C01805=1100.666,-5.311,447.503,176.248,14.221,151.801
C01806=1100.661,-5.561,447.516,176.246,14.220,151.802
C01807=1100.655,-5.810,447.530,176.244,14.220,151.802
C01808=1100.649,-6.060,447.543,176.242,14.219,151.803
C01809=1100.643,-6.309,447.557,176.240,14.219,151.803
C01810=1100.637,-6.559,447.571,176.238,14.218,151.803
C01811=1100.631,-6.808,447.584,176.236,14.218,151.804
C01812=1100.626,-7.058,447.597,176.234,14.218,151.804
C01813=1100.620,-7.307,447.610,176.232,14.217,151.804
C01814=1100.614,-7.557,447.624,176.230,14.216,151.805
C01815=1100.608,-7.806,447.637,176.228,14.216,151.805
C01816=1100.602,-8.055,447.651,176.225,14.215,151.805
C01817=1100.597,-8.306,447.664,176.223,14.214,151.806
C01818=1100.590,-8.555,447.677,176.221,14.214,151.806
C01819=1100.585,-8.804,447.691,176.219,14.213,151.807
C01820=1100.578,-9.054,447.705,176.217,14.213,151.807
C01821=1100.573,-9.305,447.718,176.215,14.212,151.807
C01822=1100.567,-9.554,447.731,176.213,14.211,151.808
C01823=1100.561,-9.804,447.745,176.210,14.211,151.808
C01824=1100.555,-10.053,447.758,176.208,14.211,151.808
C01825=1100.550,-10.303,447.771,176.206,14.210,151.809
C01826=1100.544,-10.552,447.785,176.204,14.210,151.809
C01827=1100.537,-10.801,447.798,176.202,14.209,151.809
C01828=1100.532,-11.052,447.811,176.200,14.209,151.810
C01829=1100.526,-11.301,447.824,176.198,14.208,151.810
C01830=1100.521,-11.551,447.838,176.195,14.207,151.810
C01831=1100.515,-11.800,447.851,176.193,14.206,151.811
C01832=1100.509,-12.050,447.864,176.191,14.206,151.811
C01833=1100.503,-12.299,447.878,176.189,14.205,151.811
C01834=1100.498,-12.548,447.890,176.187,14.205,151.812
C01835=1100.492,-12.798,447.904,176.185,14.204,151.812
C01836=1100.486,-13.047,447.917,176.183,14.204,151.813
C01837=1100.480,-13.297,447.930,176.181,14.203,151.813
C01838=1100.475,-13.547,447.944,176.179,14.203,151.813
C01839=1100.468,-13.796,447.957,176.177,14.202,151.813
C01840=1100.463,-14.046,447.970,176.175,14.201,151.814
C01841=1100.457,-14.295,447.983,176.173,14.201,151.814
C01842=1100.451,-14.545,447.996,176.171,14.200,151.815
C01843=1100.446,-14.795,448.010,176.169,14.200,151.815
C01844=1100.440,-15.045,448.022,176.167,14.199,151.815
C01845=1100.434,-15.294,448.035,176.165,14.198,151.816
C01846=1100.428,-15.544,448.049,176.163,14.198,151.816
C01847=1100.422,-15.794,448.062,176.160,14.197,151.816
C01848=1100.416,-16.061,448.076,176.158,14.196,151.817
C01849=1100.409,-16.328,448.090,176.156,14.196,151.817
C01850=1100.403,-16.596,448.104,176.154,14.195,151.817
C01851=1100.397,-16.863,448.118,176.152,14.195,151.818
C01852=1100.391,-17.113,448.131,176.150,14.194,151.818
C01853=1100.385,-17.362,448.144,176.148,14.194,151.818
C01854=1100.379,-17.612,448.157,176.145,14.194,151.819
C01855=1100.373,-17.861,448.170,176.144,14.193,151.819
C01856=1100.367,-18.111,448.183,176.141,14.193,151.820
C01857=1100.362,-18.360,448.196,176.140,14.192,151.820
C01858=1100.356,-18.610,448.209,176.137,14.191,151.820
C01859=1100.350,-18.859,448.222,176.135,14.190,151.821
C01860=1100.344,-19.109,448.235,176.133,14.190,151.821
C01861=1100.338,-19.358,448.248,176.131,14.189,151.821
C01862=1100.333,-19.609,448.261,176.128,14.189,151.822
C01863=1100.327,-19.858,448.274,176.127,14.188,151.822
C01864=1100.321,-20.108,448.287,176.125,14.187,151.822
C01865=1100.315,-20.358,448.299,176.123,14.187,151.823
C01866=1100.309,-20.607,448.313,176.121,14.186,151.823
C01867=1100.303,-20.857,448.325,176.118,14.186,151.823
C01868=1100.298,-21.106,448.339,176.117,14.185,151.824
C01869=1100.292,-21.356,448.351,176.114,14.185,151.824
C01870=1100.286,-21.606,448.364,176.113,14.184,151.824
C01871=1100.280,-21.855,448.377,176.110,14.184,151.825
C01872=1100.274,-22.105,448.390,176.108,14.183,151.825
C01873=1100.268,-22.354,448.403,176.106,14.183,151.825
C01874=1100.262,-22.604,448.416,176.104,14.182,151.826
C01875=1100.257,-22.853,448.428,176.102,14.181,151.826
C01876=1100.251,-23.103,448.442,176.100,14.181,151.826
C01877=1100.245,-23.352,448.454,176.098,14.180,151.827
C01878=1100.239,-23.602,448.467,176.096,14.180,151.827
C01879=1100.233,-23.852,448.480,176.094,14.179,151.827
C01880=1100.227,-24.101,448.492,176.092,14.178,151.828
C01881=1100.221,-24.351,448.505,176.090,14.178,151.828
C01882=1100.215,-24.600,448.518,176.088,14.177,151.828
C01883=1100.210,-24.850,448.531,176.086,14.177,151.829
C01884=1100.204,-25.100,448.544,176.084,14.176,151.829
C01885=1100.198,-25.350,448.556,176.082,14.176,151.829
C01886=1100.192,-25.599,448.569,176.080,14.175,151.830
C01887=1100.187,-25.848,448.582,176.078,14.174,151.830
C01888=1100.181,-26.098,448.594,176.076,14.174,151.830
C01889=1100.175,-26.348,448.607,176.074,14.173,151.831
C01890=1100.169,-26.597,448.620,176.072,14.173,151.831
C01891=1100.163,-26.847,448.633,176.070,14.172,151.831
C01892=1100.158,-27.096,448.645,176.068,14.172,151.832
C01893=1100.152,-27.346,448.657,176.066,14.171,151.832
C01894=1100.146,-27.596,448.671,176.064,14.170,151.832
C01895=1100.140,-27.845,448.683,176.062,14.170,151.833
C01896=1100.134,-28.095,448.696,176.060,14.169,151.833
C01897=1100.128,-28.345,448.708,176.058,14.169,151.833
C01898=1100.123,-28.594,448.720,176.056,14.168,151.834
C01899=1100.116,-28.844,448.734,176.054,14.168,151.834
C01900=1100.110,-29.094,448.746,176.052,14.167,151.834
C01901=1100.105,-29.343,448.759,176.050,14.166,151.835
C01902=1100.099,-29.593,448.771,176.048,14.166,151.835
C01903=1100.093,-29.842,448.784,176.046,14.165,151.835
C01904=1100.087,-30.092,448.796,176.044,14.165,151.836
C01905=1100.080,-30.341,448.809,176.042,14.164,151.836
C01906=1100.075,-30.591,448.821,176.040,14.164,151.836
C01907=1100.069,-30.841,448.834,176.038,14.163,151.837
C01908=1100.063,-31.090,448.846,176.036,14.162,151.837
C01909=1100.057,-31.340,448.859,176.034,14.162,151.837
C01910=1100.052,-31.590,448.871,176.032,14.161,151.838
C01911=1100.046,-31.840,448.884,176.030,14.161,151.838
C01912=1100.039,-32.106,448.896,176.028,14.160,151.838
C01913=1100.033,-32.372,448.911,176.026,14.160,151.839
C01914=1100.026,-32.639,448.924,176.024,14.159,151.839
C01915=1100.021,-32.906,448.937,176.022,14.158,151.839
C01916=1100.015,-33.156,448.950,176.020,14.158,151.840
C01917=1100.008,-33.405,448.962,176.018,14.157,151.840
C01918=1100.003,-33.654,448.974,176.016,14.157,151.840
C01919=1099.997,-33.904,448.986,176.014,14.156,151.841
C01920=1099.991,-34.154,448.999,176.012,14.156,151.841
C01921=1099.985,-34.404,449.011,176.010,14.155,151.841
C01922=1099.980,-34.653,449.024,176.008,14.154,151.842
C01923=1099.973,-34.903,449.036,176.006,14.154,151.842
C01924=1099.967,-35.153,449.048,176.004,14.153,151.842
C01925=1099.962,-35.402,449.060,176.002,14.153,151.843
C01926=1099.956,-35.652,449.073,176.000,14.152,151.843
C01927=1099.950,-35.902,449.085,175.998,14.152,151.843
C01928=1099.944,-36.152,449.098,175.996,14.151,151.844
C01929=1099.938,-36.400,449.110,175.994,14.151,151.844
C01930=1099.932,-36.650,449.122,175.993,14.150,151.844
C01931=1099.927,-36.900,449.135,175.991,14.150,151.844
C01932=1099.921,-37.149,449.147,175.989,14.149,151.845
C01933=1099.915,-37.399,449.159,175.987,14.148,151.845
C01934=1099.909,-37.649,449.172,175.985,14.148,151.845
C01935=1099.903,-37.898,449.184,175.983,14.147,151.846
C01936=1099.897,-38.148,449.196,175.981,14.147,151.846
C01937=1099.892,-38.398,449.209,175.978,14.146,151.847
C01938=1099.887,-38.648,449.220,175.977,14.146,151.847
C01939=1099.880,-38.897,449.232,175.975,14.145,151.847
C01940=1099.874,-39.147,449.245,175.973,14.144,151.848
C01941=1099.869,-39.396,449.257,175.971,14.144,151.848
C01942=1099.862,-39.646,449.269,175.969,14.143,151.848
C01943=1099.856,-39.896,449.281,175.967,14.143,151.848
C01944=1099.851,-40.145,449.294,175.965,14.142,151.849
C01945=1099.844,-40.394,449.306,175.963,14.142,151.849
C01946=1099.838,-40.644,449.318,175.961,14.141,151.849
C01947=1099.833,-40.894,449.330,175.959,14.141,151.850
C01948=1099.827,-41.144,449.342,175.957,14.140,151.850
C01949=1099.821,-41.394,449.354,175.956,14.140,151.850
C01950=1099.815,-41.643,449.366,175.953,14.139,151.851
C01951=1099.809,-41.892,449.378,175.951,14.139,151.851
C01952=1099.803,-42.142,449.391,175.950,14.138,151.851
C01953=1099.797,-42.392,449.402,175.947,14.137,151.852
C01954=1099.791,-42.642,449.414,175.945,14.137,151.852
C01955=1099.785,-42.891,449.427,175.943,14.136,151.852
C01956=1099.779,-43.140,449.438,175.941,14.136,151.853
C01957=1099.773,-43.390,449.451,175.940,14.135,151.853
C01958=1099.768,-43.641,449.463,175.938,14.135,151.853
C01959=1099.762,-43.890,449.474,175.936,14.134,151.854
C01960=1099.756,-44.139,449.487,175.934,14.134,151.854
C01961=1099.750,-44.388,449.498,175.932,14.133,151.854
C01962=1099.744,-44.639,449.510,175.930,14.133,151.855
C01963=1099.738,-44.889,449.523,175.928,14.132,151.855
C01964=1099.732,-45.138,449.534,175.926,14.131,151.855
C01965=1099.726,-45.387,449.547,175.924,14.131,151.856
C01966=1099.720,-45.638,449.558,175.922,14.130,151.856
C01967=1099.715,-45.887,449.570,175.920,14.130,151.856
C01968=1099.708,-46.136,449.582,175.919,14.130,151.856
C01969=1099.703,-46.386,449.594,175.917,14.129,151.857
C01970=1099.697,-46.636,449.606,175.915,14.128,151.857
C01971=1099.691,-46.885,449.618,175.913,14.128,151.858
C01972=1099.685,-47.135,449.630,175.911,14.127,151.858
C01973=1099.679,-47.385,449.642,175.909,14.127,151.858
C01974=1099.673,-47.634,449.654,175.907,14.126,151.859
C01975=1099.667,-47.884,449.665,175.905,14.126,151.859
C01976=1099.661,-48.151,449.678,175.903,14.125,151.859
C01977=1099.655,-48.419,449.691,175.901,14.124,151.859
C01978=1099.649,-48.685,449.704,175.899,14.124,151.860
C01979=1099.643,-48.952,449.716,175.897,14.123,151.860
C01980=1099.637,-49.202,449.728,175.895,14.123,151.860
C01981=1099.630,-49.451,449.740,175.893,14.122,151.861
C01982=1099.625,-49.701,449.752,175.892,14.122,151.861
C01983=1099.618,-49.951,449.764,175.890,14.121,151.861
C01984=1099.613,-50.200,449.775,175.888,14.121,151.862
C01985=1099.607,-50.450,449.787,175.886,14.120,151.862
C01986=1099.601,-50.699,449.799,175.884,14.120,151.862
C01987=1099.595,-50.949,449.811,175.882,14.119,151.863
C01988=1099.589,-51.198,449.822,175.880,14.119,151.863
C01989=1099.583,-51.449,449.834,175.878,14.118,151.863
C01990=1099.577,-51.698,449.846,175.877,14.118,151.864
C01991=1099.571,-51.948,449.857,175.875,14.117,151.864
C01992=1099.565,-52.198,449.870,175.873,14.117,151.864
C01993=1099.559,-52.447,449.881,175.871,14.116,151.865
C01994=1099.553,-52.697,449.892,175.868,14.116,151.865
C01995=1099.546,-52.946,449.904,175.867,14.115,151.865
C01996=1099.541,-53.196,449.916,175.865,14.114,151.866
C01997=1099.534,-53.446,449.928,175.863,14.115,151.866
C01998=1099.529,-53.695,449.939,175.861,14.114,151.866
C01999=1099.523,-53.945,449.951,175.859,14.114,151.867
C02000=1099.517,-54.195,449.962,175.857,14.113,151.867
C02001=1099.510,-54.444,449.974,175.855,14.112,151.867
C02002=1099.505,-54.694,449.985,175.853,14.112,151.868
C02003=1099.499,-54.944,449.997,175.851,14.111,151.868
C02004=1099.492,-55.194,450.009,175.850,14.111,151.868
C02005=1099.486,-55.443,450.020,175.848,14.111,151.869
C02006=1099.481,-55.693,450.032,175.846,14.110,151.869
C02007=1099.475,-55.942,450.044,175.844,14.110,151.869
C02008=1099.468,-56.192,450.055,175.842,14.109,151.870
C02009=1099.462,-56.441,450.067,175.840,14.109,151.870
C02010=1099.457,-56.692,450.078,175.839,14.108,151.870
C02011=1099.451,-56.941,450.089,175.837,14.108,151.870
C02012=1099.444,-57.191,450.101,175.835,14.107,151.871
C02013=1099.439,-57.440,450.112,175.833,14.107,151.871
C02014=1099.433,-57.690,450.125,175.831,14.106,151.872
C02015=1099.427,-57.939,450.136,175.829,14.106,151.872
C02016=1099.421,-58.190,450.147,175.828,14.105,151.872
C02017=1099.415,-58.438,450.158,175.825,14.105,151.872
C02018=1099.408,-58.689,450.170,175.824,14.104,151.873
C02019=1099.403,-58.938,450.182,175.821,14.104,151.873
C02020=1099.397,-59.188,450.193,175.820,14.103,151.873
C02021=1099.391,-59.438,450.204,175.818,14.103,151.874
C02022=1099.384,-59.687,450.216,175.816,14.103,151.874
C02023=1099.379,-59.937,450.227,175.814,14.102,151.874
C02024=1099.373,-60.187,450.239,175.812,14.102,151.875
C02025=1099.367,-60.436,450.250,175.810,14.101,151.875
C02026=1099.361,-60.685,450.261,175.808,14.100,151.875
C02027=1099.355,-60.936,450.272,175.807,14.101,151.876
C02028=1099.349,-61.185,450.284,175.805,14.100,151.876
C02029=1099.343,-61.435,450.296,175.803,14.099,151.876
C02030=1099.337,-61.685,450.307,175.801,14.099,151.877
C02031=1099.331,-61.934,450.319,175.799,14.098,151.877
C02032=1099.325,-62.184,450.329,175.798,14.098,151.877
C02033=1099.319,-62.434,450.341,175.796,14.098,151.878
C02034=1099.314,-62.684,450.352,175.794,14.097,151.878
C02035=1099.308,-62.932,450.364,175.792,14.097,151.878
C02036=1099.301,-63.183,450.375,175.790,14.096,151.879
C02037=1099.296,-63.432,450.386,175.788,14.095,151.879
C02038=1099.289,-63.682,450.397,175.787,14.095,151.879
C02039=1099.283,-63.931,450.409,175.785,14.095,151.879
C02040=1099.278,-64.200,450.421,175.783,14.094,151.880
C02041=1099.271,-64.468,450.433,175.781,14.094,151.880
C02042=1099.264,-64.736,450.446,175.778,14.093,151.881
C02043=1099.258,-65.005,450.457,175.777,14.093,151.881
C02044=1099.252,-65.254,450.468,175.775,14.092,151.881
C02045=1099.246,-65.504,450.479,175.773,14.092,151.882
C02046=1099.240,-65.754,450.490,175.771,14.091,151.882
C02047=1099.235,-66.003,450.502,175.769,14.091,151.882
C02048=1099.228,-66.253,450.514,175.767,14.090,151.883
C02049=1099.223,-66.503,450.525,175.765,14.090,151.883
C02050=1099.217,-66.752,450.535,175.764,14.090,151.883
C02051=1099.210,-67.002,450.547,175.762,14.089,151.883
C02052=1099.205,-67.252,450.558,175.760,14.088,151.884
C02053=1099.198,-67.501,450.570,175.758,14.088,151.884
C02054=1099.192,-67.751,450.580,175.757,14.088,151.884
C02055=1099.187,-68.000,450.591,175.755,14.088,151.885
C02056=1099.181,-68.251,450.603,175.753,14.087,151.885
C02057=1099.175,-68.500,450.614,175.751,14.086,151.885
C02058=1099.170,-68.750,450.625,175.749,14.086,151.886
C02059=1099.163,-69.000,450.636,175.748,14.086,151.886
C02060=1099.157,-69.250,450.647,175.746,14.085,151.886
C02061=1099.152,-69.499,450.658,175.744,14.085,151.887
C02062=1099.145,-69.749,450.670,175.742,14.084,151.887
C02063=1099.139,-69.998,450.681,175.741,14.084,151.887
C02064=1099.134,-70.248,450.692,175.738,14.083,151.888
C02065=1099.128,-70.497,450.702,175.737,14.083,151.888
C02066=1099.121,-70.747,450.714,175.734,14.082,151.888
C02067=1099.116,-70.997,450.725,175.733,14.082,151.889
C02068=1099.110,-71.246,450.735,175.731,14.081,151.889
C02069=1099.104,-71.496,450.747,175.729,14.081,151.889
C02070=1099.098,-71.746,450.758,175.727,14.080,151.889
C02071=1099.093,-71.996,450.769,175.725,14.080,151.890
C02072=1099.087,-72.245,450.780,175.724,14.080,151.890
C02073=1099.081,-72.495,450.791,175.722,14.079,151.890
C02074=1099.075,-72.745,450.802,175.720,14.078,151.891
C02075=1099.069,-72.994,450.813,175.718,14.078,151.891
C02076=1099.063,-73.245,450.824,175.717,14.078,151.891
C02077=1099.057,-73.494,450.835,175.715,14.077,151.892
C02078=1099.052,-73.744,450.846,175.713,14.077,151.892
C02079=1099.046,-73.993,450.857,175.711,14.076,151.892
C02080=1099.039,-74.243,450.868,175.710,14.077,151.893
C02081=1099.034,-74.493,450.879,175.708,14.076,151.893
C02082=1099.028,-74.742,450.890,175.706,14.075,151.893
C02083=1099.022,-74.991,450.900,175.704,14.075,151.894
C02084=1099.015,-75.242,450.911,175.703,14.075,151.894
C02085=1099.009,-75.491,450.922,175.700,14.074,151.894
C02086=1099.004,-75.741,450.933,175.698,14.074,151.895
C02087=1098.997,-75.991,450.944,175.697,14.074,151.895
C02088=1098.992,-76.240,450.955,175.695,14.073,151.895
C02089=1098.986,-76.490,450.966,175.693,14.072,151.896
C02090=1098.979,-76.740,450.977,175.691,14.072,151.896
C02091=1098.973,-76.990,450.987,175.690,14.072,151.896
C02092=1098.968,-77.239,450.998,175.688,14.072,151.897
C02093=1098.962,-77.489,451.009,175.686,14.071,151.897
C02094=1098.956,-77.739,451.020,175.685,14.071,151.897
C02095=1098.950,-77.988,451.031,175.683,14.071,151.898
C02096=1098.943,-78.238,451.041,175.681,14.070,151.898
C02097=1098.938,-78.487,451.052,175.678,14.070,151.898
C02098=1098.931,-78.737,451.063,175.677,14.069,151.898
C02099=1098.926,-78.987,451.074,175.675,14.069,151.899
C02100=1098.920,-79.237,451.084,175.673,14.068,151.899
C02101=1098.914,-79.486,451.095,175.672,14.068,151.899
C02102=1098.907,-79.736,451.106,175.670,14.068,151.900
C02103=1098.902,-79.986,451.117,175.668,14.067,151.900
C02104=1098.895,-80.256,451.129,175.666,14.067,151.901
C02105=1098.889,-80.527,451.140,175.664,14.066,151.901
C02106=1098.882,-80.797,451.151,175.663,14.066,151.901
C02107=1098.875,-81.068,451.163,175.660,14.066,151.902
C02108=1098.870,-81.318,451.174,175.658,14.065,151.902
C02109=1098.863,-81.567,451.184,175.656,14.065,151.902
C02110=1098.857,-81.817,451.195,175.655,14.065,151.903
C02111=1098.851,-82.066,451.206,175.653,14.065,151.903
C02112=1098.845,-82.316,451.216,175.651,14.064,151.903
C02113=1098.839,-82.566,451.227,175.650,14.064,151.904
C02114=1098.832,-82.816,451.237,175.648,14.064,151.904
C02115=1098.826,-83.065,451.248,175.646,14.063,151.904
C02116=1098.821,-83.315,451.258,175.644,14.063,151.905
C02117=1098.814,-83.564,451.269,175.643,14.062,151.905
C02118=1098.808,-83.815,451.280,175.640,14.062,151.905
C02119=1098.802,-84.064,451.291,175.639,14.062,151.906
C02120=1098.796,-84.314,451.300,175.637,14.062,151.906
C02121=1098.790,-84.563,451.311,175.635,14.061,151.906
C02122=1098.784,-84.814,451.322,175.634,14.061,151.907
C02123=1098.778,-85.063,451.333,175.632,14.061,151.907
C02124=1098.772,-85.313,451.343,175.630,14.060,151.907
C02125=1098.766,-85.562,451.353,175.629,14.060,151.908
C02126=1098.760,-85.811,451.364,175.626,14.060,151.908
C02127=1098.754,-86.062,451.375,175.625,14.059,151.908
C02128=1098.748,-86.311,451.385,175.623,14.059,151.909
C02129=1098.742,-86.561,451.396,175.621,14.059,151.909
C02130=1098.735,-86.810,451.406,175.619,14.058,151.909
C02131=1098.730,-87.060,451.416,175.618,14.058,151.910
C02132=1098.724,-87.310,451.427,175.616,14.058,151.910
C02133=1098.717,-87.560,451.438,175.614,14.057,151.910
C02134=1098.712,-87.810,451.448,175.612,14.058,151.911
C02135=1098.705,-88.059,451.458,175.610,14.057,151.911
C02136=1098.699,-88.308,451.469,175.608,14.057,151.911
C02137=1098.693,-88.559,451.480,175.607,14.056,151.912
C02138=1098.687,-88.808,451.490,175.605,14.056,151.912
C02139=1098.681,-89.058,451.500,175.603,14.055,151.912
C02140=1098.675,-89.308,451.510,175.602,14.056,151.913
C02141=1098.669,-89.557,451.521,175.600,14.055,151.913
C02142=1098.663,-89.807,451.531,175.598,14.055,151.913
C02143=1098.657,-90.056,451.542,175.596,14.055,151.914
C02144=1098.651,-90.307,451.552,175.594,14.054,151.914
C02145=1098.645,-90.556,451.562,175.593,14.054,151.914
C02146=1098.639,-90.806,451.573,175.591,14.054,151.915
C02147=1098.633,-91.056,451.583,175.589,14.053,151.915
C02148=1098.627,-91.305,451.594,175.588,14.053,151.915
C02149=1098.621,-91.555,451.603,175.586,14.053,151.916
C02150=1098.615,-91.804,451.614,175.584,14.052,151.916
C02151=1098.608,-92.055,451.624,175.582,14.052,151.916
C02152=1098.603,-92.304,451.635,175.580,14.052,151.917
C02153=1098.596,-92.554,451.645,175.578,14.051,151.917
C02154=1098.591,-92.804,451.655,175.577,14.052,151.917
C02155=1098.584,-93.053,451.666,175.575,14.051,151.918
C02156=1098.579,-93.303,451.676,175.574,14.051,151.918
C02157=1098.573,-93.553,451.687,175.572,14.050,151.918
C02158=1098.567,-93.802,451.696,175.570,14.050,151.919
C02159=1098.561,-94.052,451.707,175.568,14.050,151.919
C02160=1098.554,-94.302,451.717,175.566,14.050,151.919
C02161=1098.549,-94.552,451.728,175.564,14.049,151.920
C02162=1098.543,-94.802,451.738,175.563,14.049,151.920
C02163=1098.537,-95.051,451.748,175.561,14.049,151.920
C02164=1098.531,-95.301,451.758,175.560,14.049,151.921
C02165=1098.525,-95.550,451.769,175.558,14.048,151.921
C02166=1098.519,-95.800,451.778,175.555,14.048,151.921
C02167=1098.513,-96.050,451.789,175.554,14.048,151.922
C02168=1098.506,-96.323,451.799,175.552,14.048,151.922
C02169=1098.500,-96.595,451.811,175.550,14.047,151.922
C02170=1098.493,-96.868,451.822,175.549,14.047,151.923
C02171=1098.486,-97.141,451.833,175.547,14.047,151.923
C02172=1098.481,-97.391,451.844,175.545,14.046,151.923
C02173=1098.474,-97.640,451.854,175.543,14.046,151.924
C02174=1098.469,-97.890,451.864,175.541,14.046,151.924
C02175=1098.463,-98.140,451.874,175.539,14.045,151.925
C02176=1098.456,-98.389,451.884,175.538,14.045,151.925
C02177=1098.451,-98.640,451.894,175.536,14.045,151.925
C02178=1098.444,-98.889,451.904,175.535,14.045,151.926
C02179=1098.438,-99.138,451.914,175.533,14.045,151.926
C02180=1098.433,-99.389,451.924,175.530,14.044,151.926
C02181=1098.426,-99.638,451.934,175.529,14.044,151.927
C02182=1098.420,-99.888,451.944,175.527,14.044,151.927
C02183=1098.413,-100.137,451.955,175.526,14.044,151.927
C02184=1098.408,-100.388,451.965,175.524,14.044,151.928
C02185=1098.401,-100.637,451.974,175.522,14.044,151.928
C02186=1098.395,-100.887,451.985,175.520,14.043,151.928
C02187=1098.389,-101.137,451.995,175.518,14.043,151.929
C02188=1098.383,-101.386,452.004,175.517,14.043,151.929
C02189=1098.377,-101.636,452.015,175.515,14.042,151.929
C02190=1098.371,-101.886,452.025,175.514,14.043,151.930
C02191=1098.365,-102.136,452.034,175.512,14.042,151.930
C02192=1098.359,-102.385,452.045,175.510,14.042,151.931
C02193=1098.353,-102.634,452.054,175.508,14.042,151.931
C02194=1098.347,-102.885,452.064,175.506,14.041,151.931
C02195=1098.341,-103.134,452.075,175.505,14.041,151.931
C02196=1098.334,-103.384,452.084,175.503,14.041,151.932
C02197=1098.329,-103.634,452.094,175.501,14.041,151.932
C02198=1098.323,-103.883,452.104,175.499,14.041,151.933
C02199=1098.316,-104.133,452.114,175.498,14.041,151.933
C02200=1098.310,-104.382,452.124,175.496,14.040,151.933
C02201=1098.305,-104.633,452.134,175.495,14.041,151.934
C02202=1098.298,-104.882,452.144,175.493,14.040,151.934
C02203=1098.292,-105.132,452.154,175.491,14.040,151.934
C02204=1098.286,-105.381,452.163,175.489,14.040,151.935
C02205=1098.280,-105.631,452.173,175.487,14.039,151.935
C02206=1098.274,-105.881,452.184,175.486,14.039,151.935
C02207=1098.268,-106.130,452.193,175.484,14.039,151.936
C02208=1098.262,-106.380,452.203,175.483,14.039,151.936
C02209=1098.256,-106.630,452.212,175.480,14.039,151.936
C02210=1098.250,-106.880,452.223,175.479,14.039,151.937
C02211=1098.244,-107.129,452.233,175.477,14.038,151.937
C02212=1098.237,-107.379,452.242,175.476,14.039,151.938
C02213=1098.231,-107.629,452.252,175.474,14.038,151.938
C02214=1098.225,-107.879,452.262,175.472,14.038,151.938
C02215=1098.219,-108.129,452.271,175.470,14.038,151.939
C02216=1098.213,-108.378,452.282,175.468,14.037,151.939
C02217=1098.207,-108.628,452.292,175.467,14.038,151.939
C02218=1098.201,-108.878,452.301,175.465,14.037,151.940
C02219=1098.195,-109.127,452.311,175.463,14.037,151.940
C02220=1098.189,-109.377,452.320,175.461,14.037,151.940
C02221=1098.182,-109.627,452.330,175.460,14.037,151.941
C02222=1098.176,-109.876,452.340,175.458,14.037,151.941
C02223=1098.170,-110.126,452.350,175.456,14.037,151.941
C02224=1098.164,-110.376,452.359,175.455,14.036,151.942
C02225=1098.158,-110.626,452.369,175.453,14.037,151.942
C02226=1098.152,-110.876,452.379,175.451,14.036,151.943
C02227=1098.146,-111.125,452.389,175.450,14.036,151.943
C02228=1098.140,-111.375,452.398,175.448,14.036,151.943
C02229=1098.133,-111.624,452.408,175.446,14.036,151.944
C02230=1098.127,-111.874,452.418,175.444,14.036,151.944
C02231=1098.121,-112.124,452.428,175.443,14.036,151.944
C02232=1098.115,-112.363,452.437,175.441,14.036,151.945
C02233=1098.109,-112.602,452.446,175.440,14.036,151.945
C02234=1098.103,-112.841,452.455,175.437,14.035,151.945
C02235=1098.098,-113.081,452.464,175.436,14.036,151.946
C02236=1098.091,-113.319,452.474,175.434,14.035,151.946
C02237=1098.085,-113.559,452.483,175.433,14.035,151.946
C02238=1098.080,-113.798,452.493,175.431,14.035,151.947
C02239=1098.073,-114.037,452.501,175.429,14.035,151.947
C02240=1098.067,-114.287,452.511,175.428,14.035,151.948
C02241=1098.062,-114.536,452.520,175.426,14.034,151.948
C02242=1098.056,-114.786,452.530,175.425,14.035,151.948
C02243=1098.049,-115.036,452.539,175.422,14.035,151.949
C02244=1098.043,-115.285,452.549,175.421,14.034,151.949
C02245=1098.037,-115.535,452.558,175.419,14.034,151.949
C02246=1098.031,-115.785,452.568,175.418,14.035,151.950
C02247=1098.025,-116.035,452.578,175.415,14.034,151.950
C02248=1098.019,-116.285,452.587,175.414,14.034,151.950
C02249=1098.012,-116.534,452.597,175.412,14.034,151.951
C02250=1098.006,-116.784,452.606,175.411,14.034,151.951
C02251=1098.000,-117.034,452.616,175.409,14.033,151.951
C02252=1097.994,-117.284,452.625,175.407,14.034,151.952
C02253=1097.988,-117.534,452.635,175.405,14.034,151.952
C02254=1097.981,-117.783,452.645,175.404,14.034,151.953
C02255=1097.975,-118.033,452.654,175.402,14.033,151.953
C02256=1097.970,-118.282,452.663,175.400,14.034,151.953
C02257=1097.964,-118.532,452.673,175.398,14.033,151.954
C02258=1097.957,-118.782,452.682,175.397,14.033,151.954
C02259=1097.951,-119.032,452.692,175.395,14.033,151.954
C02260=1097.945,-119.281,452.702,175.393,14.033,151.955
C02261=1097.939,-119.531,452.711,175.392,14.034,151.955
C02262=1097.933,-119.781,452.721,175.390,14.033,151.956
C02263=1097.926,-120.030,452.730,175.389,14.033,151.956
C02264=1097.920,-120.280,452.739,175.386,14.033,151.956
C02265=1097.914,-120.531,452.748,175.385,14.033,151.957
C02266=1097.908,-120.781,452.758,175.383,14.033,151.957
C02267=1097.902,-121.030,452.767,175.382,14.033,151.957
C02268=1097.896,-121.279,452.776,175.379,14.033,151.958
C02269=1097.890,-121.529,452.786,175.378,14.033,151.958
C02270=1097.884,-121.779,452.796,175.376,14.032,151.959
C02271=1097.877,-122.029,452.805,175.375,14.033,151.959
C02272=1097.870,-122.278,452.814,175.373,14.033,151.959
C02273=1097.864,-122.528,452.824,175.371,14.033,151.960
C02274=1097.858,-122.778,452.833,175.370,14.033,151.960
C02275=1097.853,-123.028,452.842,175.368,14.032,151.960
C02276=1097.847,-123.277,452.851,175.366,14.033,151.961
C02277=1097.840,-123.527,452.861,175.364,14.032,151.961
C02278=1097.834,-123.777,452.870,175.363,14.033,151.962
C02279=1097.827,-124.026,452.879,175.361,14.032,151.962
C02280=1097.821,-124.276,452.889,175.359,14.032,151.962
C02281=1097.815,-124.527,452.898,175.358,14.033,151.963
C02282=1097.810,-124.776,452.907,175.356,14.033,151.963
C02283=1097.804,-125.026,452.917,175.354,14.032,151.963
C02284=1097.797,-125.275,452.926,175.352,14.032,151.964
C02285=1097.791,-125.525,452.935,175.351,14.033,151.964
C02286=1097.784,-125.775,452.945,175.349,14.032,151.965
C02287=1097.779,-126.025,452.954,175.347,14.033,151.965
C02288=1097.772,-126.275,452.963,175.346,14.033,151.965
C02289=1097.765,-126.524,452.972,175.344,14.032,151.966
C02290=1097.760,-126.773,452.981,175.342,14.033,151.966
C02291=1097.754,-127.024,452.990,175.340,14.032,151.967
C02292=1097.746,-127.319,453.001,175.339,14.033,151.967
C02293=1097.739,-127.615,453.013,175.337,14.032,151.967
C02294=1097.731,-127.911,453.023,175.334,14.032,151.968
C02295=1097.726,-128.206,453.034,175.333,14.033,151.968
C02296=1097.317,-128.228,452.928,175.291,14.129,151.996
C02297=1097.321,-127.958,452.918,175.293,14.130,151.996
C02298=1097.328,-127.689,452.908,175.295,14.129,151.996
C02299=1097.335,-127.419,452.898,175.297,14.130,151.995
C02300=1097.341,-127.150,452.888,175.298,14.129,151.995
C02301=1097.347,-126.900,452.879,175.300,14.130,151.995
C02302=1097.353,-126.650,452.870,175.302,14.130,151.994
C02303=1097.359,-126.400,452.860,175.304,14.130,151.994
C02304=1097.366,-126.151,452.851,175.305,14.129,151.993
C02305=1097.372,-125.901,452.842,175.307,14.129,151.993
C02306=1097.378,-125.652,452.833,175.308,14.130,151.993
C02307=1097.384,-125.401,452.824,175.310,14.129,151.992
C02308=1097.391,-125.152,452.815,175.312,14.130,151.992
C02309=1097.397,-124.902,452.805,175.314,14.129,151.991
C02310=1097.403,-124.652,452.796,175.315,14.130,151.991
C02311=1097.409,-124.402,452.786,175.317,14.130,151.991
C02312=1097.415,-124.152,452.777,175.318,14.129,151.990
C02313=1097.421,-123.903,452.769,175.321,14.130,151.990
C02314=1097.427,-123.653,452.759,175.322,14.130,151.990
C02315=1097.434,-123.404,452.750,175.324,14.130,151.989
C02316=1097.440,-123.154,452.740,175.325,14.130,151.989
C02317=1097.446,-122.904,452.730,175.327,14.130,151.989
C02318=1097.452,-122.654,452.721,175.329,14.130,151.988
C02319=1097.458,-122.404,452.712,175.331,14.130,151.988
C02320=1097.464,-122.155,452.703,175.332,14.130,151.987
C02321=1097.470,-121.905,452.694,175.334,14.131,151.987
C02322=1097.477,-121.655,452.684,175.336,14.130,151.987
C02323=1097.483,-121.406,452.675,175.337,14.130,151.986
C02324=1097.489,-121.156,452.665,175.339,14.131,151.986
C02325=1097.495,-120.906,452.656,175.340,14.130,151.986
C02326=1097.501,-120.656,452.646,175.343,14.130,151.985
C02327=1097.508,-120.406,452.636,175.344,14.130,151.985
C02328=1097.513,-120.156,452.628,175.346,14.131,151.984
C02329=1097.520,-119.907,452.619,175.347,14.131,151.984
C02330=1097.526,-119.657,452.609,175.350,14.131,151.984
C02331=1097.532,-119.408,452.600,175.351,14.131,151.983
C02332=1097.538,-119.158,452.590,175.353,14.131,151.983
C02333=1097.544,-118.908,452.581,175.354,14.131,151.983
C02334=1097.551,-118.658,452.571,175.356,14.132,151.982
C02335=1097.557,-118.408,452.562,175.358,14.131,151.982
C02336=1097.563,-118.159,452.552,175.360,14.131,151.981
C02337=1097.569,-117.909,452.542,175.361,14.132,151.981
C02338=1097.575,-117.659,452.533,175.363,14.132,151.981
C02339=1097.581,-117.409,452.523,175.365,14.131,151.980
C02340=1097.587,-117.160,452.514,175.366,14.132,151.980
C02341=1097.593,-116.910,452.504,175.368,14.132,151.980
C02342=1097.599,-116.661,452.495,175.370,14.132,151.979
C02343=1097.605,-116.411,452.485,175.371,14.132,151.979
C02344=1097.612,-116.161,452.476,175.373,14.132,151.979
C02345=1097.618,-115.911,452.466,175.375,14.132,151.978
C02346=1097.624,-115.661,452.457,175.377,14.133,151.978
C02347=1097.630,-115.412,452.447,175.378,14.132,151.978
C02348=1097.636,-115.162,452.438,175.380,14.133,151.977
C02349=1097.643,-114.912,452.428,175.382,14.133,151.977
C02350=1097.649,-114.662,452.418,175.384,14.133,151.977
C02351=1097.655,-114.412,452.409,175.385,14.133,151.976
C02352=1097.661,-114.163,452.399,175.387,14.133,151.976
C02353=1097.667,-113.913,452.390,175.388,14.133,151.975
C02354=1097.673,-113.663,452.380,175.391,14.133,151.975
C02355=1097.679,-113.414,452.371,175.392,14.133,151.975
C02356=1097.685,-113.164,452.361,175.394,14.134,151.974
C02357=1097.691,-112.909,452.351,175.395,14.133,151.974
C02358=1097.698,-112.654,452.342,175.397,14.134,151.974
C02359=1097.704,-112.399,452.332,175.399,14.134,151.973
C02360=1097.710,-112.145,452.322,175.401,14.135,151.973
C02361=1097.716,-111.895,452.312,175.402,14.134,151.973
C02362=1097.723,-111.646,452.302,175.404,14.134,151.972
C02363=1097.729,-111.396,452.293,175.405,14.135,151.972
C02364=1097.735,-111.146,452.283,175.408,14.135,151.972
C02365=1097.741,-110.896,452.273,175.409,14.134,151.971
C02366=1097.747,-110.646,452.264,175.411,14.135,151.971
C02367=1097.753,-110.397,452.254,175.412,14.135,151.970
C02368=1097.760,-110.147,452.245,175.414,14.136,151.970
C02369=1097.765,-109.897,452.234,175.416,14.135,151.970
C02370=1097.772,-109.647,452.224,175.418,14.135,151.969
C02371=1097.778,-109.398,452.215,175.420,14.136,151.969
C02372=1097.784,-109.148,452.205,175.421,14.136,151.969
C02373=1097.790,-108.898,452.196,175.423,14.137,151.968
C02374=1097.796,-108.648,452.186,175.425,14.136,151.968
C02375=1097.803,-108.399,452.176,175.427,14.136,151.968
C02376=1097.809,-108.149,452.166,175.428,14.137,151.967
C02377=1097.815,-107.900,452.157,175.430,14.137,151.967
C02378=1097.820,-107.649,452.146,175.431,14.137,151.967
C02379=1097.827,-107.400,452.137,175.433,14.137,151.966
C02380=1097.833,-107.150,452.127,175.435,14.137,151.966
C02381=1097.839,-106.901,452.117,175.437,14.138,151.966
C02382=1097.845,-106.651,452.107,175.438,14.137,151.965
C02383=1097.851,-106.401,452.097,175.440,14.138,151.965
C02384=1097.857,-106.151,452.088,175.442,14.138,151.965
C02385=1097.864,-105.902,452.077,175.443,14.138,151.964
C02386=1097.870,-105.652,452.068,175.446,14.139,151.964
C02387=1097.876,-105.402,452.058,175.447,14.139,151.964
C02388=1097.881,-105.152,452.048,175.449,14.139,151.963
C02389=1097.888,-104.903,452.038,175.450,14.139,151.963
C02390=1097.894,-104.653,452.028,175.452,14.139,151.963
C02391=1097.900,-104.403,452.019,175.454,14.139,151.962
C02392=1097.906,-104.153,452.009,175.455,14.140,151.962
C02393=1097.912,-103.904,451.998,175.458,14.140,151.961
C02394=1097.918,-103.654,451.989,175.459,14.140,151.961
C02395=1097.924,-103.404,451.979,175.461,14.140,151.961
C02396=1097.930,-103.154,451.969,175.462,14.141,151.961
C02397=1097.936,-102.905,451.959,175.464,14.141,151.960
C02398=1097.942,-102.655,451.949,175.465,14.141,151.960
C02399=1097.949,-102.404,451.939,175.468,14.141,151.959
C02400=1097.955,-102.155,451.928,175.470,14.142,151.959
C02401=1097.961,-101.906,451.919,175.471,14.142,151.959
C02402=1097.967,-101.656,451.909,175.473,14.142,151.958
C02403=1097.973,-101.406,451.898,175.474,14.142,151.958
C02404=1097.979,-101.156,451.889,175.476,14.142,151.958
C02405=1097.985,-100.907,451.879,175.478,14.143,151.957
C02406=1097.991,-100.657,451.868,175.480,14.143,151.957
C02407=1097.997,-100.407,451.859,175.482,14.143,151.957
C02408=1098.003,-100.158,451.849,175.483,14.143,151.956
C02409=1098.009,-99.908,451.838,175.485,14.144,151.956
C02410=1098.015,-99.658,451.829,175.486,14.143,151.956
C02411=1098.022,-99.408,451.819,175.488,14.144,151.955
C02412=1098.027,-99.159,451.808,175.490,14.145,151.955
C02413=1098.033,-98.909,451.799,175.492,14.145,151.955
C02414=1098.041,-98.659,451.788,175.494,14.145,151.954
C02415=1098.047,-98.409,451.779,175.495,14.145,151.954
C02416=1098.052,-98.159,451.768,175.497,14.145,151.954
C02417=1098.059,-97.910,451.758,175.499,14.146,151.953
C02418=1098.064,-97.660,451.748,175.500,14.146,151.953
C02419=1098.071,-97.411,451.738,175.502,14.146,151.953
C02420=1098.077,-97.161,451.728,175.504,14.146,151.952
C02421=1098.083,-96.889,451.717,175.506,14.147,151.952
C02422=1098.090,-96.616,451.706,175.508,14.147,151.952
C02423=1098.096,-96.342,451.695,175.510,14.147,151.951
C02424=1098.103,-96.069,451.683,175.512,14.148,151.951
C02425=1098.109,-95.820,451.672,175.513,14.148,151.951
C02426=1098.115,-95.570,451.663,175.515,14.148,151.950
C02427=1098.120,-95.320,451.653,175.517,14.148,151.950
C02428=1098.127,-95.071,451.642,175.519,14.149,151.950
C02429=1098.132,-94.821,451.632,175.520,14.150,151.949
C02430=1098.139,-94.572,451.622,175.522,14.149,151.949
C02431=1098.144,-94.321,451.612,175.524,14.150,151.949
C02432=1098.151,-94.072,451.601,175.526,14.150,151.948
C02433=1098.156,-93.821,451.591,175.527,14.150,151.948
C02434=1098.163,-93.572,451.581,175.529,14.151,151.948
C02435=1098.168,-93.322,451.571,175.530,14.151,151.947
C02436=1098.175,-93.073,451.560,175.533,14.151,151.947
C02437=1098.180,-92.823,451.550,175.534,14.152,151.947
C02438=1098.187,-92.574,451.540,175.536,14.152,151.946
C02439=1098.192,-92.324,451.530,175.538,14.152,151.946
C02440=1098.199,-92.074,451.519,175.540,14.153,151.946
C02441=1098.204,-91.825,451.509,175.541,14.153,151.945
C02442=1098.210,-91.574,451.498,175.543,14.153,151.945
C02443=1098.217,-91.325,451.488,175.545,14.154,151.945
C02444=1098.222,-91.075,451.478,175.546,14.154,151.944
C02445=1098.229,-90.826,451.467,175.548,14.155,151.944
C02446=1098.234,-90.576,451.457,175.550,14.154,151.944
C02447=1098.241,-90.326,451.447,175.551,14.155,151.943
C02448=1098.247,-90.077,451.436,175.554,14.155,151.943
C02449=1098.253,-89.826,451.426,175.555,14.155,151.943
C02450=1098.259,-89.577,451.415,175.557,14.156,151.942
C02451=1098.264,-89.327,451.405,175.559,14.156,151.942
C02452=1098.271,-89.078,451.395,175.560,14.156,151.942
C02453=1098.277,-88.828,451.384,175.562,14.157,151.941
C02454=1098.283,-88.578,451.374,175.564,14.158,151.941
C02455=1098.289,-88.328,451.363,175.565,14.157,151.941
C02456=1098.296,-88.079,451.353,175.567,14.158,151.940
C02457=1098.301,-87.829,451.343,175.570,14.158,151.940
C02458=1098.307,-87.579,451.332,175.571,14.158,151.940
C02459=1098.313,-87.330,451.322,175.573,14.159,151.939
C02460=1098.319,-87.080,451.311,175.575,14.159,151.939
C02461=1098.326,-86.830,451.301,175.576,14.159,151.939
C02462=1098.331,-86.580,451.290,175.578,14.160,151.938
C02463=1098.337,-86.331,451.280,175.580,14.160,151.938
C02464=1098.343,-86.081,451.269,175.581,14.160,151.938
C02465=1098.350,-85.831,451.258,175.583,14.161,151.938
C02466=1098.356,-85.581,451.249,175.585,14.161,151.937
C02467=1098.362,-85.332,451.238,175.587,14.161,151.937
C02468=1098.367,-85.082,451.227,175.588,14.162,151.937
C02469=1098.374,-84.833,451.217,175.591,14.162,151.936
C02470=1098.380,-84.582,451.206,175.592,14.162,151.936
C02471=1098.386,-84.333,451.196,175.594,14.163,151.936
C02472=1098.392,-84.084,451.185,175.596,14.163,151.935
C02473=1098.398,-83.834,451.175,175.597,14.164,151.935
C02474=1098.405,-83.584,451.164,175.599,14.164,151.935
C02475=1098.410,-83.334,451.153,175.601,14.165,151.934
C02476=1098.416,-83.085,451.142,175.603,14.165,151.934
C02477=1098.422,-82.835,451.133,175.604,14.165,151.934
C02478=1098.429,-82.585,451.121,175.607,14.165,151.933
C02479=1098.434,-82.335,451.111,175.608,14.166,151.933
C02480=1098.441,-82.086,451.100,175.610,14.166,151.933
C02481=1098.447,-81.837,451.089,175.612,14.166,151.932
C02482=1098.453,-81.586,451.079,175.614,14.167,151.932
C02483=1098.459,-81.337,451.069,175.615,14.167,151.932
C02484=1098.465,-81.087,451.058,175.617,14.168,151.931
C02485=1098.472,-80.817,451.046,175.619,14.168,151.931
C02486=1098.478,-80.546,451.034,175.621,14.169,151.931
C02487=1098.485,-80.275,451.023,175.623,14.169,151.930
C02488=1098.491,-80.005,451.011,175.625,14.170,151.930
C02489=1098.497,-79.755,451.000,175.627,14.169,151.930
C02490=1098.504,-79.505,450.990,175.628,14.170,151.929
C02491=1098.510,-79.256,450.979,175.630,14.171,151.929
C02492=1098.515,-79.006,450.969,175.632,14.170,151.929
C02493=1098.521,-78.756,450.958,175.634,14.171,151.928
C02494=1098.527,-78.506,450.947,175.635,14.172,151.928
C02495=1098.534,-78.257,450.936,175.638,14.172,151.928
C02496=1098.539,-78.008,450.926,175.639,14.172,151.927
C02497=1098.546,-77.757,450.914,175.641,14.173,151.927
C02498=1098.551,-77.508,450.903,175.643,14.173,151.927
C02499=1098.557,-77.258,450.893,175.644,14.174,151.927
C02500=1098.563,-77.008,450.882,175.646,14.174,151.926
C02501=1098.570,-76.758,450.872,175.648,14.175,151.926
C02502=1098.575,-76.509,450.861,175.650,14.175,151.926
C02503=1098.581,-76.259,450.850,175.651,14.175,151.925
C02504=1098.587,-76.009,450.839,175.653,14.176,151.925
C02505=1098.593,-75.760,450.828,175.655,14.176,151.925
C02506=1098.599,-75.510,450.817,175.657,14.177,151.924
C02507=1098.605,-75.260,450.806,175.658,14.177,151.924
C02508=1098.612,-75.011,450.795,175.660,14.178,151.924
C02509=1098.617,-74.761,450.785,175.662,14.178,151.923
C02510=1098.623,-74.512,450.774,175.664,14.179,151.923
C02511=1098.630,-74.262,450.762,175.666,14.178,151.923
C02512=1098.635,-74.012,450.752,175.668,14.179,151.922
C02513=1098.641,-73.763,450.741,175.670,14.180,151.922
C02514=1098.647,-73.512,450.729,175.671,14.181,151.922
C02515=1098.653,-73.263,450.719,175.673,14.180,151.921
C02516=1098.659,-73.014,450.708,175.675,14.181,151.921
C02517=1098.665,-72.764,450.697,175.677,14.182,151.921
C02518=1098.671,-72.514,450.686,175.679,14.182,151.920
C02519=1098.677,-72.264,450.675,175.680,14.182,151.920
C02520=1098.682,-72.015,450.664,175.682,14.183,151.920
C02521=1098.688,-71.765,450.653,175.684,14.183,151.920
C02522=1098.694,-71.515,450.642,175.686,14.184,151.919
C02523=1098.699,-71.265,450.630,175.687,14.184,151.919
C02524=1098.705,-71.016,450.619,175.689,14.185,151.919
C02525=1098.712,-70.766,450.608,175.691,14.185,151.918
C02526=1098.717,-70.516,450.597,175.693,14.186,151.918
C02527=1098.723,-70.267,450.586,175.695,14.187,151.918
C02528=1098.729,-70.017,450.575,175.696,14.186,151.917
C02529=1098.735,-69.767,450.564,175.698,14.187,151.917
C02530=1098.741,-69.518,450.553,175.700,14.188,151.917
C02531=1098.747,-69.268,450.542,175.702,14.189,151.917
C02532=1098.753,-69.018,450.531,175.703,14.188,151.916
C02533=1098.759,-68.769,450.520,175.705,14.189,151.916
C02534=1098.765,-68.520,450.509,175.707,14.190,151.916
C02535=1098.771,-68.269,450.498,175.709,14.190,151.915
C02536=1098.776,-68.020,450.486,175.711,14.191,151.915
C02537=1098.782,-67.770,450.475,175.712,14.191,151.915
C02538=1098.788,-67.520,450.464,175.714,14.191,151.914
C02539=1098.794,-67.270,450.453,175.716,14.192,151.914
C02540=1098.800,-67.021,450.442,175.718,14.193,151.914
C02541=1098.806,-66.771,450.430,175.720,14.193,151.914
C02542=1098.812,-66.522,450.419,175.721,14.193,151.913
C02543=1098.818,-66.272,450.408,175.723,14.194,151.913
C02544=1098.824,-66.022,450.397,175.725,14.195,151.913
C02545=1098.830,-65.773,450.386,175.727,14.195,151.912
C02546=1098.836,-65.523,450.374,175.729,14.196,151.912
C02547=1098.841,-65.273,450.363,175.730,14.196,151.912
C02548=1098.847,-65.024,450.352,175.733,14.196,151.911
C02549=1098.854,-64.755,450.340,175.734,14.197,151.911
C02550=1098.860,-64.487,450.328,175.736,14.198,151.911
C02551=1098.866,-64.218,450.316,175.739,14.198,151.910
C02552=1098.873,-63.950,450.303,175.740,14.199,151.910
C02553=1098.879,-63.700,450.292,175.742,14.199,151.910
C02554=1098.885,-63.451,450.281,175.745,14.200,151.909
C02555=1098.891,-63.200,450.270,175.746,14.200,151.909
C02556=1098.897,-62.952,450.259,175.747,14.201,151.909
C02557=1098.903,-62.701,450.247,175.750,14.201,151.908
C02558=1098.908,-62.452,450.236,175.752,14.202,151.908
C02559=1098.915,-62.201,450.225,175.753,14.202,151.908
C02560=1098.921,-61.953,450.213,175.755,14.202,151.908
C02561=1098.927,-61.703,450.202,175.757,14.203,151.907
C02562=1098.933,-61.453,450.191,175.759,14.204,151.907
C02563=1098.938,-61.204,450.179,175.761,14.204,151.907
C02564=1098.945,-60.953,450.167,175.763,14.205,151.906
C02565=1098.950,-60.704,450.157,175.765,14.205,151.906
C02566=1098.957,-60.454,450.145,175.766,14.206,151.906
C02567=1098.963,-60.205,450.134,175.768,14.206,151.905
C02568=1098.968,-59.954,450.122,175.770,14.207,151.905
C02569=1098.974,-59.706,450.110,175.772,14.207,151.905
C02570=1098.980,-59.456,450.099,175.774,14.208,151.904
C02571=1098.986,-59.206,450.088,175.775,14.208,151.904
C02572=1098.992,-58.957,450.077,175.777,14.209,151.904
C02573=1098.998,-58.707,450.065,175.779,14.209,151.903
C02574=1099.004,-58.457,450.054,175.781,14.210,151.903
C02575=1099.010,-58.207,450.042,175.783,14.210,151.903
C02576=1099.016,-57.958,450.031,175.785,14.211,151.903
C02577=1099.022,-57.708,450.018,175.787,14.211,151.902
C02578=1099.028,-57.459,450.008,175.788,14.211,151.902
C02579=1099.034,-57.208,449.996,175.790,14.212,151.902
C02580=1099.040,-56.960,449.985,175.792,14.213,151.901
C02581=1099.046,-56.709,449.973,175.794,14.213,151.901
C02582=1099.052,-56.460,449.961,175.796,14.214,151.901
C02583=1099.058,-56.210,449.950,175.798,14.214,151.900
C02584=1099.064,-55.961,449.938,175.799,14.214,151.900
C02585=1099.070,-55.711,449.927,175.801,14.215,151.900
C02586=1099.076,-55.461,449.915,175.803,14.216,151.899
C02587=1099.082,-55.212,449.904,175.805,14.216,151.899
C02588=1099.089,-54.961,449.893,175.807,14.217,151.899
C02589=1099.094,-54.712,449.880,175.809,14.217,151.899
C02590=1099.100,-54.462,449.869,175.811,14.218,151.898
C02591=1099.106,-54.213,449.858,175.812,14.218,151.898
C02592=1099.113,-53.963,449.846,175.814,14.219,151.898
C02593=1099.118,-53.714,449.834,175.816,14.219,151.897
C02594=1099.124,-53.464,449.823,175.818,14.220,151.897
C02595=1099.131,-53.214,449.811,175.820,14.220,151.897
C02596=1099.136,-52.965,449.799,175.822,14.221,151.896
C02597=1099.143,-52.715,449.787,175.824,14.221,151.896
C02598=1099.149,-52.466,449.776,175.825,14.222,151.896
C02599=1099.155,-52.216,449.765,175.827,14.222,151.895
C02600=1099.160,-51.966,449.752,175.829,14.223,151.895
C02601=1099.167,-51.716,449.741,175.831,14.223,151.895
C02602=1099.173,-51.467,449.729,175.833,14.224,151.894
C02603=1099.178,-51.217,449.718,175.835,14.224,151.894
C02604=1099.185,-50.967,449.706,175.837,14.225,151.894
C02605=1099.191,-50.718,449.694,175.839,14.226,151.894
C02606=1099.197,-50.468,449.682,175.841,14.226,151.893
C02607=1099.203,-50.218,449.670,175.842,14.226,151.893
C02608=1099.208,-49.968,449.659,175.844,14.227,151.893
C02609=1099.215,-49.719,449.647,175.847,14.227,151.892
C02610=1099.220,-49.470,449.635,175.848,14.228,151.892
C02611=1099.226,-49.220,449.624,175.850,14.229,151.892
C02612=1099.232,-48.970,449.611,175.852,14.230,151.891
C02613=1099.238,-48.703,449.599,175.854,14.230,151.891
C02614=1099.245,-48.436,449.586,175.856,14.231,151.891
C02615=1099.251,-48.169,449.573,175.858,14.231,151.890
C02616=1099.257,-47.902,449.561,175.860,14.232,151.890
C02617=1099.263,-47.652,449.549,175.862,14.233,151.890
C02618=1099.269,-47.403,449.537,175.864,14.233,151.889
C02619=1099.274,-47.152,449.525,175.866,14.234,151.889
C02620=1099.281,-46.903,449.513,175.868,14.234,151.889
C02621=1099.286,-46.654,449.501,175.869,14.234,151.889
C02622=1099.292,-46.403,449.490,175.871,14.235,151.888
C02623=1099.298,-46.154,449.478,175.873,14.236,151.888
C02624=1099.304,-45.905,449.466,175.875,14.236,151.888
C02625=1099.310,-45.654,449.454,175.877,14.237,151.887
C02626=1099.316,-45.405,449.442,175.879,14.237,151.887
C02627=1099.322,-45.155,449.430,175.881,14.238,151.887
C02628=1099.327,-44.906,449.417,175.883,14.239,151.886
C02629=1099.334,-44.656,449.406,175.885,14.239,151.886
C02630=1099.340,-44.406,449.394,175.887,14.240,151.886
C02631=1099.346,-44.157,449.382,175.889,14.241,151.885
C02632=1099.351,-43.907,449.369,175.890,14.241,151.885
C02633=1099.356,-43.658,449.358,175.892,14.241,151.885
C02634=1099.363,-43.408,449.346,175.894,14.242,151.885
C02635=1099.369,-43.158,449.333,175.896,14.243,151.884
C02636=1099.375,-42.909,449.322,175.898,14.243,151.884
C02637=1099.381,-42.659,449.309,175.900,14.244,151.884
C02638=1099.387,-42.409,449.297,175.902,14.244,151.883
C02639=1099.393,-42.160,449.286,175.904,14.245,151.883
C02640=1099.399,-41.910,449.273,175.906,14.246,151.883
C02641=1099.404,-41.660,449.261,175.908,14.246,151.882
C02642=1099.410,-41.411,449.249,175.910,14.247,151.882
C02643=1099.416,-41.161,449.237,175.912,14.247,151.882
C02644=1099.423,-40.911,449.225,175.914,14.248,151.881
C02645=1099.428,-40.662,449.213,175.915,14.248,151.881
C02646=1099.434,-40.412,449.201,175.917,14.249,151.881
C02647=1099.441,-40.163,449.189,175.919,14.249,151.880
C02648=1099.446,-39.913,449.176,175.921,14.250,151.880
C02649=1099.452,-39.664,449.164,175.923,14.250,151.880
C02650=1099.458,-39.414,449.152,175.925,14.251,151.880
C02651=1099.463,-39.164,449.141,175.927,14.252,151.879
C02652=1099.469,-38.914,449.128,175.929,14.252,151.879
C02653=1099.476,-38.665,449.116,175.931,14.253,151.879
C02654=1099.481,-38.416,449.104,175.933,14.254,151.878
C02655=1099.487,-38.166,449.091,175.935,14.254,151.878
C02656=1099.493,-37.916,449.079,175.937,14.255,151.878
C02657=1099.498,-37.667,449.067,175.939,14.256,151.877
C02658=1099.505,-37.417,449.055,175.941,14.256,151.877
C02659=1099.511,-37.167,449.042,175.943,14.257,151.877
C02660=1099.516,-36.918,449.030,175.945,14.257,151.876
C02661=1099.522,-36.668,449.017,175.946,14.258,151.876
C02662=1099.528,-36.418,449.005,175.949,14.258,151.876
C02663=1099.534,-36.169,448.993,175.951,14.259,151.875
C02664=1099.540,-35.919,448.981,175.952,14.260,151.875
C02665=1099.546,-35.670,448.968,175.954,14.260,151.875
C02666=1099.552,-35.419,448.956,175.956,14.260,151.875
C02667=1099.557,-35.170,448.944,175.958,14.261,151.874
C02668=1099.563,-34.920,448.931,175.960,14.261,151.874
C02669=1099.569,-34.670,448.919,175.962,14.262,151.874
C02670=1099.575,-34.422,448.907,175.964,14.263,151.873
C02671=1099.581,-34.172,448.894,175.965,14.264,151.873
C02672=1099.587,-33.922,448.881,175.968,14.264,151.873
C02673=1099.593,-33.672,448.869,175.969,14.265,151.872
C02674=1099.598,-33.423,448.857,175.971,14.266,151.872
C02675=1099.604,-33.173,448.844,175.974,14.266,151.872
C02676=1099.611,-32.924,448.832,175.975,14.267,151.871
C02677=1099.616,-32.657,448.819,175.977,14.267,151.871
C02678=1099.623,-32.390,448.806,175.979,14.268,151.871
C02679=1099.629,-32.123,448.792,175.981,14.268,151.870
C02680=1099.636,-31.856,448.779,175.984,14.269,151.870
C02681=1099.642,-31.607,448.767,175.986,14.270,151.870
C02682=1099.647,-31.357,448.754,175.988,14.271,151.869
C02683=1099.653,-31.107,448.742,175.990,14.271,151.869
C02684=1099.659,-30.858,448.729,175.992,14.272,151.869
C02685=1099.665,-30.608,448.716,175.994,14.273,151.869
C02686=1099.671,-30.358,448.704,175.996,14.273,151.868
C02687=1099.676,-30.109,448.691,175.997,14.273,151.868
C02688=1099.682,-29.859,448.679,175.999,14.274,151.868
C02689=1099.688,-29.609,448.666,176.001,14.274,151.867
C02690=1099.695,-29.360,448.654,176.003,14.275,151.867
C02691=1099.701,-29.110,448.642,176.005,14.275,151.867
C02692=1099.706,-28.861,448.629,176.007,14.276,151.866
C02693=1099.712,-28.612,448.616,176.009,14.277,151.866
C02694=1099.718,-28.362,448.604,176.011,14.277,151.866
C02695=1099.724,-28.112,448.591,176.013,14.278,151.865
C02696=1099.730,-27.862,448.579,176.015,14.279,151.865
C02697=1099.735,-27.613,448.566,176.017,14.279,151.865
C02698=1099.741,-27.363,448.553,176.019,14.280,151.864
C02699=1099.747,-27.114,448.541,176.021,14.280,151.864
C02700=1099.753,-26.864,448.528,176.023,14.281,151.864
C02701=1099.759,-26.614,448.515,176.025,14.282,151.863
C02702=1099.765,-26.365,448.503,176.027,14.282,151.863
C02703=1099.771,-26.115,448.490,176.029,14.283,151.863
C02704=1099.776,-25.866,448.477,176.031,14.283,151.862
C02705=1099.783,-25.616,448.464,176.033,14.284,151.862
C02706=1099.789,-25.366,448.452,176.035,14.285,151.862
C02707=1099.793,-25.117,448.439,176.038,14.286,151.861
C02708=1099.799,-24.867,448.426,176.040,14.287,151.861
C02709=1099.805,-24.618,448.413,176.042,14.287,151.861
C02710=1099.811,-24.368,448.400,176.044,14.288,151.861
C02711=1099.817,-24.118,448.388,176.046,14.288,151.860
C02712=1099.823,-23.869,448.375,176.048,14.289,151.860
C02713=1099.829,-23.620,448.362,176.050,14.290,151.860
C02714=1099.834,-23.370,448.350,176.052,14.290,151.859
C02715=1099.840,-23.120,448.337,176.054,14.291,151.859
C02716=1099.846,-22.870,448.323,176.056,14.291,151.859
C02717=1099.852,-22.620,448.311,176.058,14.292,151.858
C02718=1099.858,-22.371,448.298,176.060,14.292,151.858
C02719=1099.864,-22.121,448.285,176.062,14.293,151.858
C02720=1099.869,-21.872,448.273,176.064,14.294,151.857
C02721=1099.875,-21.623,448.260,176.066,14.294,151.857
C02722=1099.881,-21.373,448.247,176.067,14.295,151.857
C02723=1099.887,-21.123,448.234,176.070,14.295,151.856
C02724=1099.893,-20.873,448.221,176.072,14.296,151.856
C02725=1099.899,-20.623,448.208,176.074,14.296,151.856
C02726=1099.905,-20.374,448.195,176.076,14.297,151.855
C02727=1099.911,-20.124,448.182,176.077,14.298,151.855
C02728=1099.916,-19.875,448.170,176.080,14.298,151.855
C02729=1099.922,-19.626,448.156,176.082,14.299,151.854
C02730=1099.927,-19.376,448.144,176.084,14.299,151.854
C02731=1099.934,-19.126,448.130,176.086,14.300,151.854
C02732=1099.940,-18.877,448.118,176.087,14.301,151.853
C02733=1099.946,-18.627,448.105,176.090,14.301,151.853
C02734=1099.951,-18.377,448.091,176.092,14.302,151.853
C02735=1099.957,-18.128,448.078,176.094,14.302,151.852
C02736=1099.963,-17.878,448.066,176.096,14.303,151.852
C02737=1099.969,-17.629,448.052,176.098,14.303,151.852
C02738=1099.975,-17.379,448.040,176.100,14.304,151.851
C02739=1099.981,-17.129,448.026,176.102,14.306,151.851
C02740=1099.987,-16.879,448.013,176.105,14.306,151.851
C02741=1099.993,-16.612,448.000,176.106,14.307,151.850
C02742=1099.999,-16.345,447.986,176.109,14.307,151.850
C02743=1100.006,-16.077,447.972,176.110,14.308,151.850
C02744=1100.012,-15.809,447.958,176.113,14.308,151.849
C02745=1100.017,-15.560,447.944,176.115,14.309,151.849
C02746=1100.024,-15.311,447.931,176.117,14.309,151.849
C02747=1100.030,-15.061,447.918,176.119,14.310,151.848
C02748=1100.035,-14.811,447.905,176.122,14.311,151.848
C02749=1100.041,-14.561,447.892,176.123,14.312,151.848
C02750=1100.047,-14.312,447.879,176.126,14.312,151.847
C02751=1100.052,-14.062,447.866,176.127,14.313,151.847
C02752=1100.058,-13.812,447.852,176.129,14.313,151.847
C02753=1100.065,-13.563,447.839,176.132,14.314,151.846
C02754=1100.069,-13.314,447.826,176.133,14.314,151.846
C02755=1100.075,-13.064,447.813,176.136,14.315,151.846
C02756=1100.081,-12.815,447.799,176.137,14.316,151.845
C02757=1100.087,-12.565,447.787,176.139,14.316,151.845
C02758=1100.093,-12.316,447.773,176.142,14.317,151.845
C02759=1100.098,-12.066,447.760,176.143,14.317,151.844
C02760=1100.104,-11.816,447.747,176.146,14.318,151.844
C02761=1100.110,-11.567,447.733,176.147,14.318,151.844
C02762=1100.116,-11.317,447.720,176.150,14.319,151.843
C02763=1100.121,-11.067,447.707,176.152,14.320,151.843
C02764=1100.128,-10.818,447.693,176.155,14.320,151.843
C02765=1100.134,-10.569,447.680,176.156,14.321,151.842
C02766=1100.139,-10.319,447.667,176.158,14.322,151.842
C02767=1100.145,-10.069,447.654,176.160,14.322,151.842
C02768=1100.151,-9.820,447.640,176.162,14.323,151.841
C02769=1100.157,-9.570,447.627,176.165,14.323,151.841
C02770=1100.162,-9.320,447.613,176.166,14.324,151.841
C02771=1100.168,-9.071,447.600,176.169,14.324,151.840
C02772=1100.174,-8.821,447.586,176.170,14.325,151.840
C02773=1100.180,-8.571,447.574,176.173,14.326,151.840
C02774=1100.186,-8.322,447.560,176.175,14.327,151.839
C02775=1100.191,-8.073,447.547,176.177,14.327,151.839
C02776=1100.198,-7.823,447.533,176.179,14.328,151.839
C02777=1100.204,-7.573,447.519,176.182,14.328,151.838
C02778=1100.209,-7.323,447.506,176.183,14.329,151.838
C02779=1100.215,-7.074,447.493,176.186,14.329,151.838
C02780=1100.221,-6.824,447.479,176.187,14.330,151.837
C02781=1100.227,-6.575,447.465,176.190,14.331,151.837
C02782=1100.233,-6.326,447.452,176.192,14.331,151.837
C02783=1100.238,-6.075,447.439,176.194,14.332,151.836
C02784=1100.244,-5.826,447.426,176.196,14.332,151.836
C02785=1100.250,-5.577,447.412,176.199,14.333,151.835
C02786=1100.256,-5.327,447.399,176.200,14.334,151.835
C02787=1100.261,-5.078,447.385,176.203,14.334,151.835
C02788=1100.268,-4.828,447.371,176.204,14.335,151.834
C02789=1100.273,-4.579,447.358,176.207,14.335,151.834
C02790=1100.280,-4.329,447.344,176.209,14.336,151.834
C02791=1100.285,-4.079,447.331,176.211,14.337,151.833
C02792=1100.291,-3.829,447.318,176.213,14.337,151.833
C02793=1100.297,-3.580,447.304,176.215,14.338,151.833
C02794=1100.303,-3.331,447.290,176.217,14.338,151.832
C02795=1100.308,-3.081,447.277,176.220,14.339,151.832
C02796=1100.314,-2.831,447.263,176.222,14.340,151.832
C02797=1100.319,-2.582,447.249,176.224,14.340,151.831
C02798=1100.326,-2.333,447.236,176.226,14.341,151.831
C02799=1100.331,-2.083,447.222,176.228,14.341,151.831
C02800=1100.337,-1.833,447.208,176.230,14.342,151.830
C02801=1100.343,-1.584,447.195,176.232,14.343,151.830
C02802=1100.349,-1.334,447.180,176.234,14.343,151.830
C02803=1100.354,-1.084,447.166,176.237,14.344,151.829
C02804=1100.360,-0.835,447.153,176.239,14.345,151.829
C02805=1100.366,-0.566,447.139,176.241,14.345,151.829
C02806=1100.372,-0.297,447.124,176.243,14.346,151.828
C02807=1100.379,-0.027,447.109,176.246,14.347,151.828
C02808=1100.384,0.242,447.094,176.248,14.347,151.827
C02809=1100.391,0.492,447.080,176.250,14.348,151.827
C02810=1100.396,0.741,447.066,176.252,14.348,151.827
C02811=1100.402,0.991,447.053,176.254,14.349,151.826
C02812=1100.407,1.240,447.039,176.256,14.350,151.826
C02813=1100.413,1.490,447.025,176.258,14.350,151.826
C02814=1100.419,1.739,447.012,176.261,14.351,151.825
C02815=1100.425,1.989,446.997,176.263,14.352,151.825
C02816=1100.430,2.239,446.983,176.265,14.352,151.824
C02817=1100.436,2.489,446.970,176.267,14.353,151.824
C02818=1100.442,2.737,446.956,176.269,14.353,151.824
C02819=1100.448,2.987,446.942,176.271,14.354,151.824
C02820=1100.453,3.236,446.928,176.273,14.354,151.823
C02821=1100.459,3.487,446.914,176.276,14.355,151.823
C02822=1100.465,3.736,446.900,176.278,14.356,151.822
C02823=1100.471,3.985,446.887,176.280,14.356,151.822
C02824=1100.477,4.235,446.873,176.282,14.357,151.822
C02825=1100.482,4.485,446.859,176.284,14.357,151.821
C02826=1100.488,4.734,446.844,176.287,14.358,151.821
C02827=1100.494,4.984,446.830,176.288,14.358,151.821
C02828=1100.500,5.233,446.817,176.291,14.359,151.820
C02829=1100.506,5.483,446.803,176.294,14.360,151.820
C02830=1100.511,5.732,446.789,176.295,14.360,151.819
C02831=1100.517,5.981,446.774,176.298,14.361,151.819
C02832=1100.523,6.231,446.760,176.299,14.361,151.819
C02833=1100.528,6.481,446.746,176.302,14.362,151.818
C02834=1100.535,6.730,446.733,176.304,14.362,151.818
C02835=1100.540,6.980,446.719,176.306,14.363,151.818
C02836=1100.546,7.230,446.704,176.309,14.364,151.817
C02837=1100.552,7.479,446.690,176.311,14.364,151.817
C02838=1100.557,7.729,446.677,176.313,14.365,151.817
C02839=1100.563,7.978,446.663,176.315,14.365,151.816
C02840=1100.569,8.227,446.648,176.317,14.365,151.816
C02841=1100.575,8.477,446.634,176.319,14.366,151.815
C02842=1100.581,8.727,446.621,176.322,14.367,151.815
C02843=1100.587,8.976,446.606,176.324,14.367,151.815
C02844=1100.593,9.226,446.592,176.326,14.368,151.814
C02845=1100.598,9.476,446.578,176.328,14.369,151.814
C02846=1100.604,9.725,446.563,176.330,14.369,151.813
C02847=1100.610,9.974,446.549,176.333,14.369,151.813
C02848=1100.616,10.224,446.535,176.334,14.370,151.813
C02849=1100.621,10.473,446.521,176.337,14.371,151.812
C02850=1100.628,10.723,446.507,176.340,14.371,151.812
C02851=1100.634,10.973,446.493,176.342,14.372,151.811
C02852=1100.639,11.222,446.479,176.344,14.372,151.811
C02853=1100.645,11.471,446.465,176.346,14.373,151.811
C02854=1100.650,11.721,446.451,176.348,14.373,151.810
C02855=1100.657,11.971,446.436,176.351,14.374,151.810
C02856=1100.662,12.220,446.422,176.353,14.375,151.810
C02857=1100.668,12.469,446.407,176.355,14.375,151.809
C02858=1100.674,12.719,446.393,176.357,14.375,151.809
C02859=1100.680,12.969,446.379,176.359,14.376,151.808
C02860=1100.685,13.218,446.365,176.361,14.376,151.808
C02861=1100.691,13.468,446.351,176.364,14.377,151.808
C02862=1100.697,13.717,446.336,176.366,14.378,151.807
C02863=1100.703,13.968,446.322,176.369,14.378,151.807
C02864=1100.709,14.216,446.307,176.371,14.378,151.806
C02865=1100.715,14.466,446.293,176.373,14.379,151.806
C02866=1100.720,14.715,446.279,176.375,14.379,151.806
C02867=1100.726,14.965,446.264,176.378,14.380,151.805
C02868=1100.732,15.214,446.250,176.380,14.381,151.805
C02869=1100.739,15.486,446.234,176.382,14.381,151.805
C02870=1100.744,15.757,446.219,176.385,14.382,151.804
C02871=1100.751,16.029,446.203,176.387,14.383,151.804
C02872=1100.757,16.299,446.188,176.389,14.383,151.803
C02873=1100.764,16.549,446.173,176.392,14.383,151.803
C02874=1100.769,16.799,446.159,176.394,14.384,151.802
C02875=1100.774,17.048,446.144,176.397,14.385,151.802
C02876=1100.780,17.298,446.129,176.399,14.385,151.802
C02877=1100.786,17.547,446.115,176.401,14.386,151.801
C02878=1100.792,17.796,446.101,176.403,14.386,151.801
C02879=1100.798,18.046,446.086,176.406,14.387,151.800
C02880=1100.804,18.295,446.072,176.408,14.387,151.800
C02881=1100.809,18.545,446.058,176.410,14.388,151.800
C02882=1100.815,18.795,446.042,176.412,14.388,151.799
C02883=1100.820,19.044,446.028,176.414,14.389,151.799
C02884=1100.827,19.294,446.014,176.417,14.390,151.799
C02885=1100.832,19.543,445.999,176.419,14.390,151.798
C02886=1100.838,19.792,445.984,176.422,14.390,151.798
C02887=1100.844,20.042,445.970,176.424,14.391,151.797
C02888=1100.849,20.292,445.955,176.426,14.391,151.797
C02889=1100.856,20.541,445.940,176.429,14.392,151.797
C02890=1100.861,20.791,445.926,176.431,14.393,151.796
C02891=1100.867,21.040,445.912,176.433,14.393,151.796
C02892=1100.873,21.290,445.896,176.435,14.393,151.795
C02893=1100.878,21.539,445.882,176.437,14.394,151.795
C02894=1100.884,21.788,445.868,176.440,14.395,151.795
C02895=1100.890,22.038,445.853,176.442,14.395,151.794
C02896=1100.895,22.288,445.838,176.444,14.396,151.794
C02897=1100.901,22.537,445.823,176.447,14.396,151.793
C02898=1100.907,22.786,445.809,176.449,14.396,151.793
C02899=1100.913,23.036,445.794,176.452,14.397,151.792
C02900=1100.918,23.286,445.779,176.454,14.398,151.792
C02901=1100.924,23.535,445.765,176.456,14.398,151.792
C02902=1100.930,23.785,445.750,176.458,14.399,151.791
C02903=1100.935,24.034,445.735,176.460,14.399,151.791
C02904=1100.941,24.284,445.720,176.463,14.400,151.790
C02905=1100.947,24.533,445.706,176.465,14.400,151.790
C02906=1100.953,24.783,445.690,176.468,14.401,151.790
C02907=1100.959,25.032,445.676,176.470,14.401,151.789
C02908=1100.965,25.282,445.661,176.472,14.401,151.789
C02909=1100.970,25.532,445.646,176.475,14.402,151.788
C02910=1100.976,25.781,445.631,176.477,14.402,151.788
C02911=1100.982,26.030,445.617,176.479,14.403,151.787
C02912=1100.988,26.280,445.602,176.482,14.403,151.787
C02913=1100.993,26.529,445.587,176.484,14.404,151.787
C02914=1100.999,26.778,445.572,176.487,14.404,151.786
C02915=1101.005,27.028,445.557,176.489,14.405,151.786
C02916=1101.010,27.278,445.543,176.491,14.405,151.785
C02917=1101.017,27.527,445.528,176.493,14.406,151.785
C02918=1101.022,27.776,445.513,176.496,14.407,151.785
C02919=1101.028,28.026,445.498,176.498,14.407,151.784
C02920=1101.034,28.275,445.483,176.500,14.407,151.784
C02921=1101.040,28.525,445.467,176.502,14.408,151.783
C02922=1101.046,28.775,445.453,176.505,14.409,151.783
C02923=1101.051,29.024,445.437,176.508,14.409,151.783
C02924=1101.057,29.273,445.423,176.510,14.409,151.782
C02925=1101.062,29.523,445.407,176.512,14.410,151.782
C02926=1101.068,29.772,445.393,176.514,14.410,151.781
C02927=1101.074,30.022,445.377,176.517,14.411,151.781
C02928=1101.080,30.271,445.363,176.519,14.411,151.780
C02929=1101.085,30.521,445.347,176.522,14.412,151.780
C02930=1101.091,30.770,445.332,176.524,14.412,151.780
C02931=1101.097,31.020,445.317,176.527,14.413,151.779
C02932=1101.103,31.269,445.302,176.529,14.413,151.779
C02933=1101.109,31.542,445.286,176.531,14.413,151.778
C02934=1101.115,31.814,445.269,176.534,14.414,151.778
C02935=1101.121,32.087,445.253,176.537,14.414,151.777
C02936=1101.128,32.360,445.237,176.539,14.415,151.777
C02937=1101.133,32.609,445.221,176.542,14.416,151.776
C02938=1101.139,32.859,445.206,176.544,14.416,151.776
C02939=1101.145,33.109,445.191,176.546,14.416,151.776
C02940=1101.151,33.358,445.176,176.549,14.417,151.775
C02941=1101.157,33.607,445.160,176.552,14.417,151.774
C02942=1101.162,33.856,445.145,176.554,14.417,151.774
C02943=1101.168,34.106,445.130,176.556,14.418,151.774
C02944=1101.173,34.355,445.115,176.559,14.419,151.773
C02945=1101.179,34.605,445.100,176.561,14.419,151.773
C02946=1101.185,34.855,445.084,176.563,14.419,151.772
C02947=1101.191,35.104,445.070,176.565,14.420,151.772
C02948=1101.196,35.354,445.054,176.568,14.421,151.771
C02949=1101.202,35.603,445.038,176.571,14.421,151.771
C02950=1101.208,35.852,445.023,176.573,14.421,151.770
C02951=1101.214,36.102,445.008,176.575,14.421,151.770
C02952=1101.220,36.351,444.993,176.578,14.422,151.770
C02953=1101.225,36.601,444.978,176.580,14.422,151.769
C02954=1101.231,36.851,444.962,176.583,14.423,151.769
C02955=1101.237,37.099,444.947,176.585,14.423,151.768
C02956=1101.243,37.349,444.931,176.588,14.424,151.768
C02957=1101.248,37.598,444.917,176.590,14.424,151.767
C02958=1101.254,37.848,444.901,176.592,14.424,151.767
C02959=1101.260,38.098,444.885,176.595,14.425,151.766
C02960=1101.266,38.347,444.870,176.598,14.425,151.766
C02961=1101.271,38.597,444.855,176.600,14.426,151.766
C02962=1101.277,38.847,444.839,176.602,14.426,151.765
C02963=1101.282,39.095,444.823,176.605,14.426,151.765
C02964=1101.289,39.345,444.808,176.607,14.427,151.764
C02965=1101.294,39.594,444.793,176.610,14.427,151.764
C02966=1101.300,39.844,444.778,176.612,14.428,151.763
C02967=1101.305,40.093,444.761,176.615,14.429,151.763
C02968=1101.311,40.342,444.747,176.617,14.428,151.762
C02969=1101.317,40.592,444.731,176.620,14.429,151.762
C02970=1101.323,40.842,444.715,176.622,14.429,151.761
C02971=1101.328,41.091,444.700,176.625,14.430,151.761
C02972=1101.334,41.341,444.684,176.627,14.430,151.761
C02973=1101.340,41.590,444.669,176.629,14.430,151.760
C02974=1101.345,41.839,444.654,176.632,14.431,151.760
C02975=1101.351,42.089,444.638,176.635,14.432,151.759
C02976=1101.357,42.339,444.622,176.637,14.432,151.759
C02977=1101.362,42.588,444.607,176.639,14.432,151.758
C02978=1101.369,42.837,444.591,176.642,14.433,151.758
C02979=1101.374,43.087,444.575,176.644,14.433,151.757
C02980=1101.379,43.336,444.560,176.647,14.433,151.757
C02981=1101.385,43.585,444.544,176.649,14.433,151.756
C02982=1101.391,43.835,444.528,176.652,14.434,151.756
C02983=1101.397,44.085,444.512,176.654,14.435,151.755
C02984=1101.403,44.334,444.498,176.656,14.435,151.755
C02985=1101.409,44.583,444.481,176.660,14.435,151.754
C02986=1101.414,44.833,444.466,176.662,14.436,151.754
C02987=1101.419,45.082,444.451,176.664,14.436,151.754
C02988=1101.425,45.332,444.434,176.666,14.436,151.753
C02989=1101.431,45.582,444.419,176.670,14.437,151.752
C02990=1101.436,45.830,444.403,176.672,14.437,151.752
C02991=1101.442,46.080,444.387,176.674,14.438,151.752
C02992=1101.448,46.330,444.371,176.677,14.438,151.751
C02993=1101.453,46.579,444.356,176.679,14.438,151.751
C02994=1101.459,46.828,444.340,176.682,14.439,151.750
C02995=1101.464,47.078,444.324,176.684,14.439,151.750
C02996=1101.470,47.327,444.308,176.687,14.440,151.749
C02997=1101.476,47.600,444.291,176.689,14.440,151.749
C02998=1101.482,47.873,444.273,176.693,14.440,151.748
C02999=1101.488,48.145,444.255,176.695,14.441,151.748
C03000=1101.495,48.418,444.239,176.698,14.441,151.747
C03001=1101.501,48.668,444.223,176.700,14.442,151.747
C03002=1101.505,48.917,444.207,176.703,14.441,151.746
C03003=1101.511,49.166,444.191,176.706,14.442,151.746
C03004=1101.517,49.416,444.175,176.708,14.443,151.745
C03005=1101.523,49.665,444.159,176.710,14.443,151.745
C03006=1101.528,49.914,444.144,176.713,14.444,151.744
C03007=1101.534,50.164,444.127,176.716,14.444,151.744
C03008=1101.540,50.413,444.111,176.718,14.444,151.743
C03009=1101.545,50.663,444.095,176.720,14.444,151.743
C03010=1101.551,50.912,444.079,176.723,14.445,151.742
C03011=1101.557,51.161,444.063,176.726,14.445,151.742
C03012=1101.562,51.411,444.048,176.728,14.445,151.741
C03013=1101.568,51.660,444.032,176.731,14.446,151.741
C03014=1101.574,51.910,444.015,176.733,14.446,151.740
C03015=1101.580,52.159,443.999,176.736,14.446,151.740
C03016=1101.585,52.408,443.984,176.739,14.447,151.739
C03017=1101.591,52.658,443.968,176.741,14.447,151.739
C03018=1101.597,52.907,443.951,176.744,14.447,151.738
C03019=1101.602,53.157,443.934,176.746,14.447,151.738
C03020=1101.608,53.407,443.919,176.749,14.448,151.737
C03021=1101.614,53.656,443.903,176.751,14.448,151.737
C03022=1101.619,53.905,443.887,176.754,14.448,151.736
C03023=1101.625,54.154,443.871,176.757,14.449,151.736
C03024=1101.631,54.404,443.855,176.759,14.449,151.735
C03025=1101.637,54.653,443.839,176.762,14.449,151.735
C03026=1101.643,54.903,443.823,176.765,14.450,151.734
C03027=1101.649,55.152,443.806,176.767,14.450,151.734
C03028=1101.654,55.402,443.789,176.769,14.450,151.733
C03029=1101.660,55.651,443.773,176.773,14.451,151.733
C03030=1101.665,55.900,443.758,176.775,14.451,151.732
C03031=1101.671,56.150,443.742,176.777,14.451,151.732
C03032=1101.677,56.399,443.725,176.781,14.451,151.731
C03033=1101.683,56.648,443.709,176.783,14.452,151.731
C03034=1101.689,56.898,443.693,176.785,14.452,151.730
C03035=1101.694,57.147,443.676,176.787,14.452,151.730
C03036=1101.700,57.397,443.660,176.791,14.452,151.729
C03037=1101.706,57.646,443.644,176.793,14.452,151.728
C03038=1101.712,57.896,443.628,176.795,14.453,151.728
C03039=1101.718,58.145,443.612,176.799,14.453,151.727
C03040=1101.723,58.395,443.595,176.801,14.453,151.727
C03041=1101.729,58.644,443.579,176.803,14.453,151.726
C03042=1101.735,58.894,443.562,176.807,14.454,151.726
C03043=1101.740,59.142,443.547,176.809,14.454,151.725
C03044=1101.746,59.392,443.530,176.811,14.454,151.725
C03045=1101.751,59.641,443.513,176.815,14.455,151.724
C03046=1101.757,59.891,443.497,176.817,14.455,151.724
C03047=1101.763,60.140,443.481,176.819,14.455,151.723
C03048=1101.769,60.389,443.465,176.823,14.455,151.722
C03049=1101.775,60.639,443.448,176.825,14.455,151.722
C03050=1101.780,60.888,443.432,176.827,14.456,151.721
C03051=1101.786,61.138,443.415,176.831,14.456,151.721
C03052=1101.792,61.387,443.399,176.833,14.456,151.720
C03053=1101.798,61.637,443.383,176.836,14.456,151.720
C03054=1101.803,61.886,443.366,176.839,14.457,151.719
C03055=1101.810,62.135,443.349,176.841,14.457,151.719
C03056=1101.815,62.384,443.333,176.844,14.457,151.718
C03057=1101.821,62.634,443.316,176.846,14.456,151.718
C03058=1101.827,62.883,443.300,176.849,14.457,151.717
C03059=1101.833,63.133,443.283,176.852,14.457,151.717
C03060=1101.839,63.383,443.267,176.854,14.457,151.716
C03061=1101.845,63.655,443.249,176.857,14.458,151.715
C03062=1101.852,63.927,443.231,176.861,14.458,151.715
C03063=1101.858,64.199,443.213,176.863,14.458,151.714
C03064=1101.865,64.472,443.195,176.867,14.459,151.713
C03065=1101.870,64.722,443.178,176.869,14.459,151.713
C03066=1101.876,64.971,443.161,176.872,14.458,151.712
C03067=1101.881,65.221,443.145,176.875,14.459,151.712
C03068=1101.887,65.469,443.128,176.877,14.459,151.711
C03069=1101.892,65.719,443.111,176.880,14.459,151.711
C03070=1101.898,65.968,443.094,176.883,14.460,151.710
C03071=1101.904,66.218,443.078,176.885,14.460,151.710
C03072=1101.910,66.467,443.061,176.888,14.459,151.709
C03073=1101.916,66.716,443.044,176.891,14.460,151.709
C03074=1101.921,66.966,443.028,176.893,14.460,151.708
C03075=1101.927,67.215,443.011,176.896,14.460,151.707
C03076=1101.932,67.465,442.994,176.899,14.461,151.707
C03077=1101.939,67.713,442.977,176.902,14.461,151.706
C03078=1101.944,67.963,442.961,176.904,14.461,151.706
C03079=1101.950,68.212,442.944,176.907,14.461,151.705
C03080=1101.955,68.462,442.928,176.910,14.461,151.705
C03081=1101.961,68.711,442.911,176.912,14.461,151.704
C03082=1101.967,68.961,442.893,176.915,14.462,151.703
C03083=1101.973,69.211,442.877,176.918,14.462,151.703
C03084=1101.978,69.460,442.860,176.920,14.462,151.702
C03085=1101.984,69.709,442.843,176.924,14.462,151.702
C03086=1101.990,69.959,442.826,176.926,14.462,151.701
C03087=1101.996,70.207,442.809,176.929,14.462,151.700
C03088=1102.001,70.457,442.793,176.932,14.462,151.700
C03089=1102.007,70.706,442.775,176.934,14.463,151.699
C03090=1102.013,70.955,442.759,176.937,14.463,151.699
C03091=1102.018,71.205,442.742,176.940,14.463,151.698
C03092=1102.024,71.454,442.725,176.942,14.463,151.698
C03093=1102.029,71.703,442.708,176.946,14.464,151.697
C03094=1102.035,71.953,442.690,176.948,14.464,151.696
C03095=1102.041,72.203,442.674,176.951,14.463,151.696
C03096=1102.046,72.452,442.657,176.954,14.464,151.695
C03097=1102.052,72.701,442.639,176.957,14.464,151.695
C03098=1102.058,72.951,442.623,176.959,14.464,151.694
C03099=1102.063,73.200,442.606,176.962,14.464,151.693
C03100=1102.069,73.449,442.589,176.965,14.464,151.693
C03101=1102.075,73.698,442.572,176.967,14.464,151.692
C03102=1102.081,73.948,442.555,176.971,14.465,151.692
C03103=1102.086,74.197,442.537,176.973,14.464,151.691
C03104=1102.092,74.447,442.521,176.976,14.464,151.691
C03105=1102.098,74.696,442.503,176.979,14.465,151.690
C03106=1102.103,74.945,442.486,176.981,14.465,151.689
C03107=1102.109,75.194,442.469,176.985,14.465,151.689
C03108=1102.115,75.445,442.452,176.987,14.465,151.688
C03109=1102.121,75.694,442.435,176.990,14.465,151.688
C03110=1102.126,75.943,442.418,176.993,14.466,151.687
C03111=1102.132,76.192,442.401,176.996,14.466,151.686
C03112=1102.138,76.441,442.383,176.998,14.465,151.686
C03113=1102.143,76.691,442.366,177.002,14.465,151.685
C03114=1102.150,76.940,442.349,177.004,14.465,151.684
C03115=1102.155,77.190,442.332,177.007,14.465,151.684
C03116=1102.160,77.439,442.315,177.010,14.466,151.683
C03117=1102.167,77.687,442.298,177.012,14.466,151.683
C03118=1102.172,77.938,442.280,177.016,14.466,151.682
C03119=1102.178,78.187,442.263,177.018,14.466,151.682
C03120=1102.183,78.436,442.245,177.021,14.466,151.681
C03121=1102.189,78.686,442.228,177.024,14.466,151.680
C03122=1102.195,78.934,442.211,177.027,14.466,151.680
C03123=1102.201,79.184,442.194,177.029,14.466,151.679
C03124=1102.206,79.434,442.177,177.033,14.466,151.678
C03125=1102.212,79.706,442.157,177.035,14.466,151.678
C03126=1102.218,79.979,442.139,177.039,14.466,151.677
C03127=1102.225,80.250,442.120,177.042,14.467,151.676
C03128=1102.231,80.523,442.100,177.045,14.466,151.676
C03129=1102.236,80.772,442.083,177.048,14.467,151.675
C03130=1102.242,81.021,442.066,177.051,14.467,151.675
C03131=1102.247,81.270,442.048,177.053,14.467,151.674
C03132=1102.253,81.520,442.030,177.056,14.467,151.673
C03133=1102.259,81.770,442.013,177.059,14.467,151.673
C03134=1102.264,82.019,441.996,177.062,14.467,151.672
C03135=1102.270,82.268,441.979,177.065,14.467,151.671
C03136=1102.277,82.517,441.961,177.068,14.467,151.671
C03137=1102.282,82.766,441.943,177.071,14.468,151.670
C03138=1102.287,83.016,441.927,177.074,14.467,151.669
C03139=1102.293,83.265,441.909,177.076,14.467,151.669
C03140=1102.299,83.515,441.891,177.080,14.467,151.668
C03141=1102.304,83.764,441.873,177.082,14.467,151.668
C03142=1102.310,84.013,441.856,177.085,14.467,151.667
C03143=1102.316,84.263,441.838,177.088,14.467,151.666
C03144=1102.322,84.512,441.820,177.091,14.467,151.666
C03145=1102.327,84.761,441.804,177.094,14.467,151.665
C03146=1102.332,85.010,441.786,177.097,14.467,151.664
C03147=1102.338,85.260,441.768,177.099,14.467,151.664
C03148=1102.344,85.509,441.751,177.103,14.467,151.663
C03149=1102.349,85.758,441.733,177.105,14.467,151.662
C03150=1102.356,86.008,441.715,177.108,14.467,151.662
C03151=1102.361,86.257,441.697,177.111,14.467,151.661
C03152=1102.367,86.506,441.680,177.114,14.467,151.661
C03153=1102.373,86.756,441.662,177.117,14.468,151.660
C03154=1102.378,87.005,441.644,177.120,14.467,151.659
C03155=1102.384,87.255,441.626,177.123,14.467,151.659
C03156=1102.390,87.504,441.609,177.126,14.467,151.658
C03157=1102.395,87.753,441.591,177.129,14.467,151.657
C03158=1102.402,88.002,441.573,177.132,14.468,151.657
C03159=1102.407,88.251,441.556,177.135,14.467,151.656
C03160=1102.413,88.501,441.538,177.137,14.467,151.655
C03161=1102.419,88.750,441.520,177.141,14.467,151.655
C03162=1102.424,88.999,441.503,177.143,14.467,151.654
C03163=1102.430,89.249,441.485,177.146,14.466,151.653
C03164=1102.436,89.498,441.467,177.150,14.467,151.653
C03165=1102.441,89.747,441.449,177.152,14.466,151.652
C03166=1102.447,89.997,441.431,177.156,14.467,151.651
C03167=1102.452,90.246,441.414,177.159,14.466,151.651
C03168=1102.459,90.495,441.395,177.161,14.466,151.650
C03169=1102.464,90.744,441.377,177.165,14.466,151.649
C03170=1102.470,90.994,441.359,177.167,14.466,151.649
C03171=1102.476,91.243,441.342,177.171,14.466,151.648
C03172=1102.481,91.492,441.324,177.173,14.466,151.647
C03173=1102.487,91.742,441.306,177.176,14.466,151.647
C03174=1102.492,91.991,441.288,177.179,14.466,151.646
C03175=1102.498,92.240,441.270,177.182,14.466,151.645
C03176=1102.504,92.489,441.252,177.185,14.466,151.645
C03177=1102.509,92.739,441.234,177.188,14.466,151.644
C03178=1102.515,92.989,441.216,177.191,14.466,151.643
C03179=1102.521,93.238,441.198,177.194,14.466,151.643
C03180=1102.527,93.487,441.180,177.197,14.466,151.642
C03181=1102.532,93.736,441.162,177.201,14.466,151.641
C03182=1102.537,93.985,441.144,177.203,14.466,151.641
C03183=1102.543,94.235,441.126,177.206,14.465,151.640
C03184=1102.549,94.484,441.108,177.209,14.466,151.639
C03185=1102.555,94.733,441.089,177.212,14.465,151.638
C03186=1102.560,94.982,441.072,177.216,14.465,151.638
C03187=1102.566,95.232,441.054,177.218,14.465,151.637
C03188=1102.571,95.481,441.035,177.221,14.465,151.636
C03189=1102.578,95.753,441.015,177.225,14.465,151.636
C03190=1102.584,96.026,440.996,177.228,14.465,151.635
C03191=1102.591,96.298,440.976,177.231,14.464,151.634
C03192=1102.597,96.571,440.956,177.235,14.464,151.633
C03193=1102.602,96.820,440.937,177.237,14.464,151.633
C03194=1102.608,97.069,440.920,177.241,14.464,151.632
C03195=1102.614,97.318,440.902,177.244,14.464,151.631
C03196=1102.619,97.568,440.883,177.246,14.464,151.631
C03197=1102.625,97.817,440.865,177.250,14.464,151.630
C03198=1102.631,98.066,440.846,177.252,14.463,151.629
C03199=1102.636,98.315,440.828,177.256,14.463,151.628
C03200=1102.642,98.565,440.810,177.259,14.463,151.628
C03201=1102.648,98.814,440.792,177.261,14.463,151.627
C03202=1102.653,99.064,440.774,177.265,14.463,151.626
C03203=1102.659,99.312,440.755,177.268,14.462,151.626
C03204=1102.665,99.562,440.737,177.271,14.463,151.625
C03205=1102.670,99.810,440.718,177.274,14.462,151.624
C03206=1102.677,100.060,440.701,177.277,14.462,151.623
C03207=1102.682,100.310,440.681,177.280,14.462,151.623
C03208=1102.688,100.559,440.664,177.283,14.462,151.622
C03209=1102.694,100.808,440.645,177.286,14.462,151.621
C03210=1102.699,101.057,440.627,177.289,14.462,151.621
C03211=1102.705,101.306,440.608,177.292,14.461,151.620
C03212=1102.710,101.556,440.590,177.296,14.461,151.619
C03213=1102.717,101.805,440.571,177.298,14.461,151.619
C03214=1102.722,102.055,440.553,177.302,14.461,151.618
C03215=1102.728,102.303,440.535,177.305,14.461,151.617
C03216=1102.733,102.553,440.516,177.308,14.461,151.616
C03217=1102.738,102.802,440.497,177.311,14.460,151.616
C03218=1102.745,103.051,440.479,177.314,14.460,151.615
C03219=1102.750,103.301,440.460,177.317,14.460,151.614
C03220=1102.756,103.550,440.442,177.320,14.460,151.613
C03221=1102.761,103.800,440.423,177.324,14.460,151.613
C03222=1102.767,104.048,440.405,177.327,14.459,151.612
C03223=1102.773,104.298,440.386,177.329,14.459,151.611
C03224=1102.778,104.547,440.368,177.333,14.459,151.610
C03225=1102.784,104.796,440.349,177.335,14.459,151.610
C03226=1102.790,105.045,440.330,177.339,14.459,151.609
C03227=1102.795,105.294,440.312,177.342,14.458,151.608
C03228=1102.801,105.544,440.293,177.345,14.459,151.608
C03229=1102.807,105.792,440.275,177.348,14.458,151.607
C03230=1102.812,106.042,440.256,177.351,14.458,151.606
C03231=1102.818,106.292,440.237,177.355,14.458,151.605
C03232=1102.824,106.540,440.219,177.358,14.457,151.605
C03233=1102.829,106.790,440.199,177.361,14.457,151.604
C03234=1102.835,107.039,440.181,177.364,14.457,151.603
C03235=1102.841,107.288,440.163,177.367,14.456,151.602
C03236=1102.846,107.538,440.143,177.370,14.456,151.602
C03237=1102.853,107.787,440.125,177.373,14.456,151.601
C03238=1102.857,108.036,440.106,177.377,14.456,151.600
C03239=1102.863,108.285,440.087,177.380,14.455,151.599
C03240=1102.870,108.535,440.069,177.383,14.455,151.599
C03241=1102.875,108.783,440.050,177.386,14.455,151.598
C03242=1102.880,109.033,440.030,177.389,14.454,151.597
C03243=1102.886,109.283,440.013,177.393,14.455,151.596
C03244=1102.892,109.532,439.993,177.395,14.454,151.596
C03245=1102.897,109.781,439.974,177.399,14.454,151.595
C03246=1102.904,110.030,439.956,177.402,14.454,151.594
C03247=1102.909,110.279,439.936,177.405,14.453,151.593
C03248=1102.914,110.528,439.918,177.409,14.453,151.592
C03249=1102.921,110.777,439.899,177.411,14.452,151.592
C03250=1102.927,111.027,439.880,177.415,14.452,151.591
C03251=1102.932,111.277,439.861,177.418,14.452,151.590
C03252=1102.937,111.525,439.842,177.421,14.452,151.589
C03253=1102.944,111.798,439.822,177.425,14.451,151.588
C03254=1102.950,112.070,439.801,177.428,14.451,151.588
C03255=1102.956,112.342,439.780,177.432,14.451,151.587
C03256=1102.962,112.615,439.759,177.435,14.450,151.586
C03257=1102.969,112.864,439.740,177.439,14.451,151.585
C03258=1102.974,113.113,439.721,177.441,14.450,151.584
C03259=1102.980,113.363,439.702,177.445,14.449,151.584
C03260=1102.985,113.611,439.683,177.448,14.449,151.583
C03261=1102.991,113.861,439.664,177.451,14.449,151.582
C03262=1102.997,114.110,439.645,177.455,14.449,151.581
C03263=1103.003,114.359,439.626,177.457,14.448,151.581
C03264=1103.008,114.608,439.607,177.461,14.448,151.580
C03265=1103.014,114.857,439.588,177.464,14.447,151.579
C03266=1103.019,115.107,439.568,177.467,14.447,151.578
C03267=1103.025,115.356,439.549,177.471,14.447,151.577
C03268=1103.030,115.605,439.530,177.473,14.447,151.577
C03269=1103.036,115.854,439.511,177.477,14.447,151.576
C03270=1103.041,116.104,439.492,177.480,14.446,151.575
C03271=1103.047,116.353,439.472,177.484,14.446,151.574
C03272=1103.052,116.602,439.454,177.487,14.445,151.573
C03273=1103.058,116.852,439.434,177.490,14.446,151.573
C03274=1103.064,117.100,439.414,177.493,14.445,151.572
C03275=1103.070,117.350,439.395,177.496,14.444,151.571
C03276=1103.075,117.598,439.376,177.500,14.444,151.570
C03277=1103.080,117.848,439.357,177.503,14.444,151.570
C03278=1103.086,118.097,439.338,177.507,14.443,151.569
C03279=1103.092,118.347,439.319,177.509,14.443,151.568
C03280=1103.098,118.596,439.299,177.513,14.443,151.567
C03281=1103.103,118.845,439.279,177.516,14.442,151.566
C03282=1103.109,119.094,439.260,177.519,14.442,151.565
C03283=1103.114,119.343,439.241,177.523,14.442,151.565
C03284=1103.120,119.592,439.221,177.525,14.441,151.564
C03285=1103.126,119.841,439.202,177.529,14.441,151.563
C03286=1103.132,120.091,439.183,177.532,14.440,151.562
C03287=1103.137,120.340,439.163,177.536,14.441,151.562
C03288=1103.143,120.588,439.144,177.539,14.440,151.561
C03289=1103.148,120.838,439.125,177.543,14.440,151.560
C03290=1103.153,121.088,439.105,177.546,14.439,151.559
C03291=1103.159,121.337,439.086,177.549,14.438,151.558
C03292=1103.165,121.586,439.066,177.552,14.438,151.557
C03293=1103.171,121.835,439.046,177.555,14.437,151.557
C03294=1103.176,122.085,439.027,177.559,14.438,151.556
C03295=1103.182,122.334,439.007,177.562,14.437,151.555
C03296=1103.187,122.582,438.988,177.566,14.437,151.554
C03297=1103.193,122.831,438.968,177.569,14.436,151.553
C03298=1103.199,123.080,438.949,177.572,14.436,151.552
C03299=1103.205,123.330,438.930,177.576,14.435,151.552
C03300=1103.210,123.579,438.909,177.578,14.435,151.551
C03301=1103.216,123.828,438.890,177.582,14.434,151.550
C03302=1103.222,124.077,438.870,177.585,14.434,151.549
C03303=1103.227,124.327,438.851,177.589,14.433,151.548
C03304=1103.233,124.576,438.832,177.592,14.433,151.547
C03305=1103.239,124.825,438.812,177.596,14.433,151.547
C03306=1103.245,125.074,438.792,177.599,14.432,151.546
C03307=1103.250,125.324,438.772,177.602,14.431,151.545
C03308=1103.256,125.573,438.753,177.605,14.431,151.544
C03309=1103.262,125.822,438.733,177.609,14.430,151.543
C03310=1103.267,126.071,438.713,177.613,14.430,151.542
C03311=1103.273,126.320,438.693,177.615,14.430,151.542
C03312=1103.279,126.569,438.674,177.619,14.429,151.541
C03313=1103.284,126.819,438.654,177.622,14.429,151.540
C03314=1103.290,127.068,438.634,177.626,14.429,151.539
C03315=1103.296,127.317,438.614,177.629,14.428,151.538
C03316=1103.302,127.566,438.594,177.632,14.427,151.537
C03317=1103.308,127.838,438.574,177.636,14.427,151.536
C03318=1103.314,128.110,438.551,177.640,14.426,151.535
C03319=1103.320,128.383,438.530,177.643,14.425,151.534
C03320=1103.327,128.655,438.508,177.647,14.425,151.533
C03321=1103.333,128.904,438.489,177.651,14.425,151.533
C03322=1103.338,129.154,438.468,177.654,14.424,151.532
C03323=1103.344,129.402,438.448,177.657,14.423,151.531
C03324=1103.350,129.652,438.429,177.661,14.423,151.530
C03325=1103.356,129.901,438.409,177.664,14.422,151.529
C03326=1103.361,130.150,438.388,177.668,14.422,151.528
C03327=1103.367,130.399,438.369,177.671,14.421,151.527
C03328=1103.373,130.648,438.349,177.675,14.421,151.526
C03329=1103.379,130.897,438.329,177.678,14.420,151.526
C03330=1103.384,131.147,438.308,177.682,14.420,151.525
C03331=1103.390,131.396,438.289,177.685,14.419,151.524
C03332=1103.396,131.645,438.269,177.688,14.418,151.523
C03333=1103.401,131.894,438.249,177.692,14.418,151.522
C03334=1103.407,132.143,438.229,177.695,14.417,151.521
C03335=1103.413,132.392,438.209,177.699,14.417,151.520
C03336=1103.418,132.641,438.189,177.702,14.416,151.519
C03337=1103.424,132.890,438.169,177.706,14.416,151.519
C03338=1103.430,133.139,438.148,177.709,14.415,151.518
C03339=1103.435,133.389,438.129,177.713,14.415,151.517
C03340=1103.441,133.638,438.109,177.716,14.414,151.516
C03341=1103.447,133.887,438.088,177.719,14.413,151.515
C03342=1103.453,134.136,438.068,177.723,14.413,151.514
C03343=1103.458,134.385,438.048,177.726,14.412,151.513
C03344=1103.464,134.634,438.028,177.730,14.412,151.512
C03345=1103.470,134.883,438.007,177.733,14.411,151.512
C03346=1103.475,135.133,437.988,177.737,14.411,151.511
C03347=1103.480,135.382,437.967,177.740,14.410,151.510
C03348=1103.486,135.631,437.947,177.744,14.410,151.509
C03349=1103.492,135.880,437.927,177.747,14.409,151.508
C03350=1103.498,136.129,437.907,177.751,14.409,151.507
C03351=1103.504,136.378,437.886,177.754,14.408,151.506
C03352=1103.510,136.627,437.866,177.757,14.407,151.505
C03353=1103.515,136.876,437.846,177.761,14.407,151.504
C03354=1103.521,137.125,437.826,177.764,14.406,151.503
C03355=1103.526,137.374,437.805,177.768,14.406,151.502
C03356=1103.532,137.623,437.785,177.771,14.405,151.502
C03357=1103.538,137.873,437.764,177.775,14.405,151.501
C03358=1103.544,138.122,437.744,177.778,14.404,151.500
C03359=1103.549,138.371,437.724,177.782,14.404,151.499
C03360=1103.554,138.620,437.703,177.785,14.403,151.498
C03361=1103.560,138.869,437.683,177.789,14.402,151.497
C03362=1103.566,139.119,437.662,177.792,14.401,151.496
C03363=1103.572,139.367,437.642,177.795,14.401,151.495
C03364=1103.578,139.617,437.622,177.799,14.400,151.494
C03365=1103.583,139.866,437.601,177.802,14.399,151.493
C03366=1103.589,140.114,437.581,177.806,14.399,151.493
C03367=1103.595,140.364,437.560,177.810,14.398,151.491
C03368=1103.601,140.613,437.540,177.814,14.398,151.491
C03369=1103.606,140.862,437.519,177.817,14.397,151.490
C03370=1103.611,141.111,437.498,177.821,14.396,151.489
C03371=1103.617,141.360,437.478,177.824,14.395,151.488
C03372=1103.623,141.609,437.458,177.828,14.395,151.487
C03373=1103.629,141.858,437.437,177.831,14.394,151.486
C03374=1103.634,142.108,437.416,177.835,14.394,151.485
C03375=1103.640,142.356,437.396,177.838,14.393,151.484
C03376=1103.646,142.606,437.375,177.841,14.392,151.483
C03377=1103.651,142.855,437.354,177.845,14.392,151.482
C03378=1103.657,143.104,437.334,177.848,14.391,151.481
C03379=1103.662,143.353,437.314,177.852,14.391,151.480
C03380=1103.668,143.601,437.293,177.856,14.389,151.479
C03381=1103.674,143.874,437.270,177.860,14.389,151.478
C03382=1103.680,144.146,437.247,177.864,14.388,151.477
C03383=1103.686,144.419,437.225,177.867,14.388,151.476
C03384=1103.694,144.691,437.202,177.871,14.387,151.475
C03385=1103.699,144.940,437.181,177.875,14.387,151.474
C03386=1103.704,145.189,437.161,177.879,14.385,151.473
C03387=1103.710,145.437,437.140,177.882,14.384,151.473
C03388=1103.716,145.687,437.119,177.886,14.384,151.472
C03389=1103.722,145.936,437.099,177.889,14.383,151.471
C03390=1103.727,146.185,437.077,177.893,14.383,151.470
C03391=1103.733,146.434,437.057,177.896,14.382,151.469
C03392=1103.738,146.684,437.036,177.900,14.381,151.468
C03393=1103.744,146.932,437.015,177.904,14.380,151.467
C03394=1103.750,147.182,436.994,177.907,14.380,151.466
C03395=1103.756,147.431,436.974,177.911,14.379,151.465
C03396=1103.761,147.679,436.953,177.915,14.379,151.464
C03397=1103.767,147.929,436.932,177.918,14.378,151.463
C03398=1103.773,148.178,436.910,177.922,14.377,151.462
C03399=1103.778,148.427,436.890,177.925,14.376,151.461
C03400=1103.785,148.676,436.869,177.929,14.375,151.460
C03401=1103.790,148.925,436.848,177.933,14.375,151.459
C03402=1103.796,149.173,436.827,177.936,14.374,151.458
C03403=1103.801,149.423,436.806,177.940,14.373,151.457
C03404=1103.807,149.671,436.785,177.943,14.372,151.456
C03405=1103.813,149.921,436.764,177.947,14.372,151.455
C03406=1103.818,150.170,436.743,177.951,14.371,151.454
C03407=1103.824,150.419,436.722,177.955,14.370,151.453
C03408=1103.830,150.668,436.700,177.958,14.369,151.452
C03409=1103.835,150.917,436.680,177.962,14.369,151.451
C03410=1103.841,151.166,436.659,177.965,14.368,151.450
C03411=1103.847,151.416,436.638,177.969,14.368,151.449
C03412=1103.852,151.664,436.616,177.972,14.367,151.449
C03413=1103.858,151.914,436.595,177.977,14.366,151.447
C03414=1103.863,152.162,436.574,177.980,14.365,151.447
C03415=1103.869,152.411,436.553,177.984,14.364,151.445
C03416=1103.875,152.661,436.532,177.987,14.364,151.445
C03417=1103.880,152.909,436.511,177.991,14.362,151.443
C03418=1103.887,153.158,436.489,177.995,14.362,151.443
C03419=1103.892,153.408,436.469,177.998,14.361,151.442
C03420=1103.897,153.656,436.447,178.002,14.360,151.441
C03421=1103.904,153.905,436.426,178.005,14.360,151.440
C03422=1103.909,154.154,436.405,178.009,14.359,151.439
C03423=1103.914,154.404,436.383,178.013,14.358,151.438
C03424=1103.920,154.652,436.362,178.017,14.357,151.437
C03425=1103.926,154.902,436.341,178.020,14.356,151.436
C03426=1103.931,155.151,436.319,178.024,14.356,151.435
C03427=1103.937,155.400,436.298,178.027,14.355,151.434
C03428=1103.943,155.649,436.276,178.032,14.354,151.433
C03429=1103.949,155.898,436.256,178.035,14.353,151.432
C03430=1103.954,156.147,436.234,178.039,14.353,151.431
C03431=1103.961,156.396,436.213,178.043,14.351,151.430
C03432=1103.965,156.645,436.191,178.047,14.351,151.429
C03433=1103.972,156.894,436.169,178.050,14.350,151.428
C03434=1103.977,157.143,436.149,178.053,14.349,151.427
C03435=1103.982,157.392,436.127,178.057,14.348,151.426
C03436=1103.989,157.641,436.106,178.061,14.347,151.425
C03437=1103.994,157.889,436.084,178.065,14.347,151.424
C03438=1104.000,158.139,436.062,178.068,14.345,151.422
C03439=1104.006,158.388,436.041,178.072,14.345,151.422
C03440=1104.011,158.637,436.020,178.076,14.344,151.420
C03441=1104.017,158.886,435.998,178.080,14.344,151.420
C03442=1104.022,159.135,435.976,178.083,14.342,151.419
C03443=1104.028,159.384,435.955,178.087,14.342,151.417
C03444=1104.034,159.633,435.934,178.091,14.341,151.417
C03445=1104.040,159.905,435.910,178.095,14.340,151.415
C03446=1104.046,160.177,435.886,178.099,14.339,151.414
C03447=1104.053,160.449,435.862,178.103,14.338,151.413
C03448=1104.059,160.721,435.839,178.107,14.337,151.412
C03449=1104.065,160.969,435.818,178.111,14.336,151.411
C03450=1104.070,161.219,435.795,178.115,14.335,151.410
C03451=1104.076,161.468,435.774,178.118,14.334,151.409
C03452=1104.082,161.716,435.753,178.122,14.334,151.408
C03453=1104.087,161.966,435.730,178.126,14.332,151.407
C03454=1104.093,162.214,435.709,178.130,14.332,151.406
C03455=1104.098,162.464,435.687,178.133,14.331,151.405
C03456=1104.104,162.712,435.666,178.137,14.330,151.404
C03457=1104.109,162.962,435.643,178.141,14.329,151.403
C03458=1104.115,163.210,435.622,178.145,14.329,151.402
C03459=1104.120,163.460,435.600,178.148,14.327,151.401
C03460=1104.126,163.708,435.579,178.152,14.327,151.400
C03461=1104.132,163.958,435.557,178.156,14.326,151.399
C03462=1104.137,164.207,435.535,178.160,14.325,151.398
C03463=1104.143,164.456,435.513,178.163,14.324,151.397
C03464=1104.149,164.705,435.490,178.167,14.324,151.396
C03465=1104.154,164.953,435.469,178.171,14.322,151.395
C03466=1104.159,165.203,435.447,178.175,14.322,151.393
C03467=1104.164,165.451,435.425,178.179,14.320,151.392
C03468=1104.170,165.701,435.403,178.183,14.320,151.391
C03469=1104.176,165.950,435.381,178.186,14.319,151.390
C03470=1104.182,166.198,435.359,178.190,14.318,151.389
C03471=1104.187,166.448,435.337,178.194,14.317,151.388
C03472=1104.193,166.696,435.316,178.198,14.316,151.387
C03473=1104.198,166.946,435.294,178.201,14.316,151.386
C03474=1104.205,167.194,435.271,178.205,14.315,151.385
C03475=1104.209,167.443,435.249,178.209,14.314,151.384
C03476=1104.216,167.692,435.228,178.213,14.313,151.383
C03477=1104.221,167.942,435.205,178.217,14.312,151.382
C03478=1104.226,168.190,435.183,178.221,14.311,151.381
C03479=1104.232,168.439,435.161,178.224,14.310,151.380
C03480=1104.238,168.689,435.139,178.228,14.310,151.379
C03481=1104.244,168.936,435.117,178.232,14.308,151.378
C03482=1104.249,169.186,435.095,178.236,14.308,151.377
C03483=1104.254,169.436,435.073,178.240,14.306,151.376
C03484=1104.260,169.683,435.051,178.244,14.306,151.375
C03485=1104.266,169.933,435.028,178.247,14.304,151.374
C03486=1104.272,170.182,435.007,178.252,14.304,151.372
C03487=1104.277,170.430,434.984,178.255,14.303,151.371
C03488=1104.283,170.680,434.962,178.259,14.302,151.370
C03489=1104.289,170.928,434.940,178.263,14.301,151.369
C03490=1104.294,171.178,434.917,178.266,14.299,151.368
C03491=1104.299,171.427,434.895,178.271,14.299,151.367
C03492=1104.306,171.675,434.873,178.274,14.297,151.366
C03493=1104.311,171.925,434.851,178.278,14.297,151.365
C03494=1104.317,172.174,434.828,178.282,14.296,151.364
C03495=1104.322,172.422,434.807,178.286,14.295,151.363
C03496=1104.328,172.671,434.784,178.289,14.294,151.362
C03497=1104.334,172.921,434.761,178.294,14.293,151.361
C03498=1104.340,173.169,434.739,178.297,14.292,151.360
C03499=1104.345,173.418,434.717,178.301,14.291,151.358
C03500=1104.351,173.667,434.694,178.305,14.290,151.357
C03501=1104.357,173.916,434.672,178.309,14.289,151.356
C03502=1104.362,174.165,434.650,178.313,14.288,151.355
C03503=1104.368,174.414,434.627,178.317,14.287,151.354
C03504=1104.374,174.662,434.606,178.321,14.286,151.353
C03505=1104.380,174.911,434.583,178.325,14.285,151.352
C03506=1104.385,175.161,434.560,178.329,14.284,151.351
C03507=1104.391,175.410,434.537,178.333,14.283,151.350
C03508=1104.397,175.658,434.515,178.336,14.282,151.349
C03509=1104.403,175.930,434.490,178.341,14.281,151.347
C03510=1104.409,176.202,434.466,178.345,14.280,151.346
C03511=1104.415,176.473,434.441,178.349,14.278,151.345
C03512=1104.422,176.745,434.417,178.354,14.278,151.344
C03513=1104.428,176.994,434.394,178.358,14.277,151.343
C03514=1104.433,177.242,434.372,178.362,14.275,151.341
C03515=1104.438,177.491,434.349,178.366,14.275,151.340
C03516=1104.445,177.740,434.327,178.369,14.273,151.339
C03517=1104.450,177.989,434.304,178.374,14.272,151.338
C03518=1104.456,178.238,434.281,178.377,14.271,151.337
C03519=1104.462,178.487,434.259,178.381,14.270,151.336
C03520=1104.467,178.736,434.236,178.385,14.269,151.335
C03521=1104.473,178.985,434.213,178.389,14.268,151.334
C03522=1104.479,179.234,434.191,178.393,14.267,151.333
C03523=1104.485,179.483,434.168,178.397,14.266,151.331
C03524=1104.490,179.731,434.146,178.401,14.265,151.330
C03525=1104.496,179.980,434.123,178.405,14.263,151.329
C03526=1104.501,180.229,434.100,178.409,14.263,151.328
C03527=1104.507,180.478,434.077,178.413,14.261,151.327
C03528=1104.514,180.727,434.055,178.417,14.260,151.326
C03529=1104.519,180.976,434.032,178.421,14.259,151.325
C03530=1104.525,181.224,434.009,178.425,14.258,151.323
C03531=1104.531,181.474,433.986,178.429,14.257,151.322
C03532=1104.536,181.723,433.964,178.433,14.256,151.321
C03533=1104.542,181.972,433.941,178.437,14.255,151.320
C03534=1104.548,182.221,433.918,178.441,14.254,151.319
C03535=1104.553,182.470,433.895,178.445,14.252,151.318
C03536=1104.560,182.718,433.872,178.449,14.252,151.317
C03537=1104.566,182.967,433.849,178.453,14.250,151.315
C03538=1104.571,183.216,433.826,178.457,14.250,151.314
C03539=1104.577,183.465,433.804,178.461,14.248,151.313
C03540=1104.583,183.714,433.781,178.465,14.247,151.312
C03541=1104.589,183.963,433.758,178.469,14.246,151.311
C03542=1104.594,184.211,433.735,178.473,14.245,151.310
C03543=1104.600,184.460,433.712,178.477,14.244,151.309
C03544=1104.606,184.709,433.689,178.481,14.243,151.307
C03545=1104.612,184.958,433.666,178.485,14.242,151.306
C03546=1104.618,185.206,433.642,178.489,14.240,151.305
C03547=1104.623,185.455,433.619,178.493,14.239,151.304
C03548=1104.629,185.704,433.596,178.498,14.238,151.303
C03549=1104.635,185.953,433.573,178.501,14.237,151.302
C03550=1104.640,186.202,433.550,178.505,14.236,151.301
C03551=1104.645,186.451,433.527,178.509,14.235,151.299
C03552=1104.651,186.700,433.504,178.513,14.234,151.298
C03553=1104.657,186.949,433.481,178.517,14.232,151.297
C03554=1104.663,187.198,433.458,178.521,14.232,151.296
C03555=1104.668,187.447,433.434,178.525,14.231,151.295
C03556=1104.674,187.695,433.411,178.529,14.230,151.294
C03557=1104.679,187.944,433.388,178.533,14.228,151.293
C03558=1104.685,188.193,433.365,178.538,14.227,151.291
C03559=1104.690,188.442,433.341,178.541,14.226,151.290
C03560=1104.696,188.691,433.318,178.546,14.225,151.289
C03561=1104.702,188.940,433.295,178.549,14.224,151.288
C03562=1104.708,189.188,433.272,178.554,14.223,151.287
C03563=1104.713,189.438,433.248,178.557,14.222,151.286
C03564=1104.719,189.686,433.225,178.562,14.221,151.284
C03565=1104.724,189.935,433.202,178.565,14.220,151.283
C03566=1104.730,190.184,433.179,178.570,14.219,151.282
C03567=1104.735,190.433,433.155,178.573,14.217,151.281
C03568=1104.741,190.681,433.132,178.578,14.216,151.280
C03569=1104.748,190.931,433.108,178.581,14.215,151.279
C03570=1104.753,191.180,433.085,178.586,14.214,151.277
C03571=1104.759,191.428,433.061,178.590,14.213,151.276
C03572=1104.764,191.677,433.038,178.594,14.212,151.275
C03573=1104.771,191.948,433.013,178.598,14.210,151.274
C03574=1104.776,192.220,432.987,178.603,14.209,151.273
C03575=1104.782,192.491,432.961,178.607,14.208,151.271
C03576=1104.789,192.762,432.936,178.612,14.207,151.270
C03577=1104.794,193.010,432.912,178.615,14.206,151.269
C03578=1104.800,193.259,432.889,178.620,14.205,151.268
C03579=1104.806,193.508,432.865,178.624,14.203,151.266
C03580=1104.811,193.757,432.841,178.628,14.202,151.265
C03581=1104.817,194.006,432.818,178.632,14.201,151.264
C03582=1104.823,194.255,432.795,178.637,14.200,151.263
C03583=1104.828,194.504,432.771,178.640,14.199,151.262
C03584=1104.834,194.752,432.747,178.645,14.198,151.261
C03585=1104.840,195.001,432.723,178.648,14.196,151.259
C03586=1104.846,195.250,432.700,178.653,14.195,151.258
C03587=1104.852,195.499,432.676,178.657,14.194,151.257
C03588=1104.857,195.748,432.653,178.661,14.193,151.256
C03589=1104.863,195.996,432.629,178.665,14.191,151.255
C03590=1104.868,196.245,432.606,178.669,14.191,151.254
C03591=1104.875,196.494,432.581,178.673,14.189,151.252
C03592=1104.880,196.743,432.558,178.678,14.188,151.251
C03593=1104.886,196.992,432.534,178.681,14.186,151.250
C03594=1104.892,197.240,432.511,178.686,14.186,151.249
C03595=1104.897,197.489,432.487,178.690,14.184,151.247
C03596=1104.903,197.738,432.463,178.694,14.183,151.246
C03597=1104.909,197.987,432.439,178.698,14.182,151.245
C03598=1104.914,198.236,432.416,178.703,14.181,151.244
C03599=1104.920,198.484,432.392,178.706,14.179,151.243
C03600=1104.926,198.733,432.368,178.711,14.178,151.241
C03601=1104.931,198.982,432.344,178.714,14.177,151.240
C03602=1104.937,199.231,432.320,178.719,14.176,151.239
C03603=1104.943,199.480,432.296,178.723,14.174,151.238
C03604=1104.949,199.728,432.272,178.727,14.173,151.237
C03605=1104.954,199.977,432.249,178.731,14.172,151.235
C03606=1104.960,200.226,432.225,178.736,14.171,151.234
C03607=1104.966,200.475,432.200,178.739,14.169,151.233
C03608=1104.972,200.723,432.177,178.744,14.168,151.232
C03609=1104.977,200.972,432.152,178.748,14.167,151.230
C03610=1104.984,201.222,432.129,178.752,14.166,151.229
C03611=1104.989,201.470,432.105,178.756,14.164,151.228
C03612=1104.995,201.718,432.081,178.761,14.163,151.227
C03613=1105.001,201.968,432.056,178.765,14.162,151.226
C03614=1105.006,202.216,432.032,178.769,14.161,151.224
C03615=1105.012,202.465,432.009,178.773,14.159,151.223
C03616=1105.018,202.714,431.984,178.778,14.158,151.222
C03617=1105.024,202.962,431.960,178.781,14.156,151.221
C03618=1105.029,203.211,431.937,178.786,14.156,151.219
C03619=1105.035,203.461,431.912,178.789,14.154,151.218
C03620=1105.041,203.709,431.888,178.794,14.153,151.217
C03621=1105.047,203.957,431.864,178.798,14.152,151.216
C03622=1105.052,204.207,431.840,178.802,14.151,151.215
C03623=1105.058,204.455,431.815,178.806,14.149,151.213
C03624=1105.064,204.704,431.792,178.811,14.148,151.212
C03625=1105.070,204.953,431.767,178.815,14.147,151.211
C03626=1105.075,205.201,431.743,178.819,14.146,151.210
C03627=1105.080,205.450,431.719,178.823,14.144,151.208
